P[294]{
   GP1:
	UF : 1, UT : 1,		CONFIG : 'N U T, 0, 0, 0',
	X =  2685.132  mm,	Y =   201.280  mm,	Z =   305.695  mm,
	W =    -3.830 deg,	P =   -10.878 deg,	R =   -17.892 deg
   GP2:
	UF : 1, UT : 1,
	J1=    90.000 deg,	J2=   135.000 deg
};
P[295]{
   GP1:
	UF : 1, UT : 1,		CONFIG : 'N U T, 0, 0, 0',
	X =  2753.412  mm,	Y =   160.459  mm,	Z =   180.671  mm,
	W =     2.791 deg,	P =    -7.674 deg,	R =   -18.462 deg
   GP2:
	UF : 1, UT : 1,
	J1=    90.000 deg,	J2=   135.000 deg
};
P[296]{
   GP1:
	UF : 1, UT : 1,		CONFIG : 'N U T, 0, 0, 0',
	X =  2867.805  mm,	Y =   160.634  mm,	Z =   182.471  mm,
	W =     9.502 deg,	P =   -26.582 deg,	R =   -20.495 deg
   GP2:
	UF : 1, UT : 1,
	J1=    89.999 deg,	J2=   135.000 deg
};
P[297]{
   GP1:
	UF : 1, UT : 1,		CONFIG : 'N U T, 0, 0, 0',
	X =  2663.741  mm,	Y =   157.782  mm,	Z =   292.643  mm,
	W =    13.374 deg,	P =   -35.036 deg,	R =   -22.495 deg
   GP2:
	UF : 1, UT : 1,
	J1=    90.000 deg,	J2=   135.000 deg
};
P[298]{
   GP1:
	UF : 1, UT : 1,		CONFIG : 'N U T, 0, 0, 0',
	X =  2363.741  mm,	Y =   272.782  mm,	Z =   292.643  mm,
	W =     -.090 deg,	P =    -5.498 deg,	R =      .950 deg
   GP2:
	UF : 1, UT : 1,
	J1=    90.000 deg,	J2=   135.000 deg
};
P[299]{
   GP1:
	UF : 1, UT : 1,		CONFIG : 'N U T, 0, 0, 0',
	X =  2378.956  mm,	Y =   265.120  mm,	Z =    86.366  mm,
	W =     1.850 deg,	P =     -.182 deg,	R =      .942 deg
   GP2:
	UF : 1, UT : 1,
	J1=    90.000 deg,	J2=   135.000 deg
};
P[300]{
   GP1:
	UF : 1, UT : 1,		CONFIG : 'N U T, 0, 0, 0',
	X =  2754.391  mm,	Y =   263.612  mm,	Z =    86.366  mm,
	W =     1.733 deg,	P =    -7.250 deg,	R =      .949 deg
   GP2:
	UF : 1, UT : 1,
	J1=    90.000 deg,	J2=   135.000 deg
};
P[301]{
   GP1:
	UF : 1, UT : 1,		CONFIG : 'N U T, 0, 0, 0',
	X =  2718.394  mm,	Y =   243.937  mm,	Z =   215.203  mm,
	W =     -.140 deg,	P =    -8.465 deg,	R =      .956 deg
   GP2:
	UF : 1, UT : 1,
	J1=    90.000 deg,	J2=   135.000 deg
};
P[302]{
   GP1:
	UF : 1, UT : 1,		CONFIG : 'N U T, 0, 0, 0',
	X =  2303.751  mm,	Y =   260.223  mm,	Z =   215.203  mm,
	W =     -.140 deg,	P =    -8.465 deg,	R =      .956 deg
   GP2:
	UF : 1, UT : 1,
	J1=    90.000 deg,	J2=   135.000 deg
};
P[303]{
   GP1:
	UF : 1, UT : 1,		CONFIG : 'N U T, 0, 0, 0',
	X =  1858.037  mm,	Y =   423.080  mm,	Z =   600.917  mm,
	W =     -.140 deg,	P =    -8.465 deg,	R =   -19.002 deg
   GP2:
	UF : 1, UT : 1,
	J1=    90.000 deg,	J2=   135.000 deg
};
P[304]{
   GP1:
	UF : 1, UT : 1,		CONFIG : 'N U T, 0, 0, 0',
	X =  1858.037  mm,	Y =   423.080  mm,	Z =   369.489  mm,
	W =    39.110 deg,	P =     2.688 deg,	R =   -82.797 deg
   GP2:
	UF : 1, UT : 1,
	J1=    90.000 deg,	J2=    90.000 deg
};
P[305]{
   GP1:
	UF : 1, UT : 1,		CONFIG : 'N U T, 0, 0, 0',
	X =  2035.037  mm,	Y =    99.189  mm,	Z =    92.489  mm,
	W =    39.110 deg,	P =     2.688 deg,	R =   -82.797 deg
   GP2:
	UF : 1, UT : 1,
	J1=    90.000 deg,	J2=    90.000 deg
};
P[306]{
   GP1:
	UF : 1, UT : 1,		CONFIG : 'N U T, 0, 0, 0',
	X =  2068.312  mm,	Y =   107.394  mm,	Z =   -18.582  mm,
	W =    37.933 deg,	P =    17.387 deg,	R =   -97.672 deg
   GP2:
	UF : 1, UT : 1,
	J1=    90.000 deg,	J2=    90.000 deg
};
P[307]{
   GP1:
	UF : 1, UT : 1,		CONFIG : 'N U T, 0, 0, 0',
	X =  2109.723  mm,	Y =    72.505  mm,	Z =   -21.222  mm,
	W =    37.933 deg,	P =    17.387 deg,	R =  -104.287 deg
   GP2:
	UF : 1, UT : 1,
	J1=    90.000 deg,	J2=    90.000 deg
};
P[308]{
   GP1:
	UF : 1, UT : 1,		CONFIG : 'N U T, 0, 0, -1',
	X =  2115.592  mm,	Y =    62.473  mm,	Z =   -16.026  mm,
	W =    44.181 deg,	P =    21.261 deg,	R =  -126.963 deg
   GP2:
	UF : 1, UT : 1,
	J1=    90.000 deg,	J2=    90.000 deg
};
P[309]{
   GP1:
	UF : 1, UT : 1,		CONFIG : 'N U T, 0, 0, -1',
	X =  2027.388  mm,	Y =   105.837  mm,	Z =    81.683  mm,
	W =    40.362 deg,	P =    21.867 deg,	R =  -139.995 deg
   GP2:
	UF : 1, UT : 1,
	J1=    90.000 deg,	J2=    90.000 deg
};
P[310]{
   GP1:
	UF : 1, UT : 1,		CONFIG : 'N U T, 0, 0, 0',
	X =  1658.817  mm,	Y =   448.694  mm,	Z =    81.684  mm,
	W =   -42.959 deg,	P =    14.926 deg,	R =    16.534 deg
   GP2:
	UF : 1, UT : 1,
	J1=    90.000 deg,	J2=    90.000 deg
};
P[311]{
   GP1:
	UF : 1, UT : 1,		CONFIG : 'N U T, 0, 0, 0',
	X =  1681.875  mm,	Y =   114.694  mm,	Z =    81.683  mm,
	W =   -42.959 deg,	P =    14.926 deg,	R =    16.534 deg
   GP2:
	UF : 1, UT : 1,
	J1=    90.000 deg,	J2=    90.000 deg
};
P[312]{
   GP1:
	UF : 1, UT : 1,		CONFIG : 'N U T, 0, 0, 0',
	X =  1685.743  mm,	Y =    59.810  mm,	Z =   -17.917  mm,
	W =   -42.807 deg,	P =    15.441 deg,	R =    16.037 deg
   GP2:
	UF : 1, UT : 1,
	J1=    90.000 deg,	J2=    90.000 deg
};
P[313]{
   GP1:
	UF : 1, UT : 1,		CONFIG : 'N U T, 0, 0, 0',
	X =  1652.429  mm,	Y =    58.946  mm,	Z =   -19.364  mm,
	W =   -42.810 deg,	P =    15.442 deg,	R =    16.034 deg
   GP2:
	UF : 1, UT : 1,
	J1=    90.000 deg,	J2=    90.000 deg
};
P[314]{
   GP1:
	UF : 1, UT : 1,		CONFIG : 'N U T, 0, 0, 0',
	X =  1640.987  mm,	Y =    56.683  mm,	Z =   -21.519  mm,
	W =   -42.181 deg,	P =    15.522 deg,	R =    -8.109 deg
   GP2:
	UF : 1, UT : 1,
	J1=    90.000 deg,	J2=    90.000 deg
};
P[315]{
   GP1:
	UF : 1, UT : 1,		CONFIG : 'N U T, 0, 0, 0',
	X =  1637.701  mm,	Y =    59.485  mm,	Z =   -19.665  mm,
	W =   -38.593 deg,	P =    25.218 deg,	R =   -16.905 deg
   GP2:
	UF : 1, UT : 1,
	J1=    90.000 deg,	J2=    90.000 deg
};
P[316]{
   GP1:
	UF : 1, UT : 1,		CONFIG : 'N U T, 0, 0, 0',
	X =  1608.736  mm,	Y =    83.348  mm,	Z =   -24.399  mm,
	W =   -38.593 deg,	P =    25.219 deg,	R =   -16.905 deg
   GP2:
	UF : 1, UT : 1,
	J1=    90.000 deg,	J2=    90.000 deg
};
P[317]{
   GP1:
	UF : 1, UT : 1,		CONFIG : 'N U T, 0, 0, 0',
	X =  1585.662  mm,	Y =   101.135  mm,	Z =   -21.859  mm,
	W =   -45.000 deg,	P =    -3.170 deg,	R =      .426 deg
   GP2:
	UF : 1, UT : 1,
	J1=    90.000 deg,	J2=    90.000 deg
};
P[318]{
   GP1:
	UF : 1, UT : 1,		CONFIG : 'N U T, 0, 0, 0',
	X =  1556.810  mm,	Y =    69.060  mm,	Z =   -21.622  mm,
	W =   -45.449 deg,	P =    19.944 deg,	R =    98.982 deg
   GP2:
	UF : 1, UT : 1,
	J1=    90.000 deg,	J2=    90.000 deg
};
P[319]{
   GP1:
	UF : 1, UT : 1,		CONFIG : 'N U T, 0, 0, 0',
	X =  1551.240  mm,	Y =    28.811  mm,	Z =   -19.922  mm,
	W =   -45.337 deg,	P =    20.062 deg,	R =    97.887 deg
   GP2:
	UF : 1, UT : 1,
	J1=    90.000 deg,	J2=    90.000 deg
};
P[320]{
   GP1:
	UF : 1, UT : 1,		CONFIG : 'N U T, 0, 0, 0',
	X =  1551.443  mm,	Y =    22.198  mm,	Z =   -20.367  mm,
	W =   -45.343 deg,	P =    20.068 deg,	R =    97.646 deg
   GP2:
	UF : 1, UT : 1,
	J1=    90.000 deg,	J2=    90.000 deg
};
P[321]{
   GP1:
	UF : 1, UT : 1,		CONFIG : 'N U T, 0, 0, 0',
	X =  1549.407  mm,	Y =    21.768  mm,	Z =   -17.950  mm,
	W =   -41.210 deg,	P =    19.947 deg,	R =    34.862 deg
   GP2:
	UF : 1, UT : 1,
	J1=    90.000 deg,	J2=    90.000 deg
};
P[322]{
   GP1:
	UF : 1, UT : 1,		CONFIG : 'N U T, 0, 0, 0',
	X =  1540.684  mm,	Y =    20.490  mm,	Z =   -17.846  mm,
	W =   -41.215 deg,	P =    19.945 deg,	R =    34.866 deg
   GP2:
	UF : 1, UT : 1,
	J1=    90.000 deg,	J2=    90.000 deg
};
P[323]{
   GP1:
	UF : 1, UT : 1,		CONFIG : 'N U T, 0, 0, 0',
	X =  1231.677  mm,	Y =   199.953  mm,	Z =   178.712  mm,
	W =   -41.215 deg,	P =    19.944 deg,	R =    40.052 deg
   GP2:
	UF : 1, UT : 1,
	J1=    90.000 deg,	J2=    90.000 deg
};
P[324]{
   GP1:
	UF : 1, UT : 1,		CONFIG : 'N U T, 0, 0, 0',
	X =   877.425  mm,	Y =  1334.354  mm,	Z =    94.527  mm,
	W =     -.178 deg,	P =    -1.186 deg,	R =    26.509 deg
   GP2:
	UF : 1, UT : 1,
	J1=    90.000 deg,	J2=    90.000 deg
};
P[325]{
   GP1:
	UF : 1, UT : 1,		CONFIG : 'N U T, 0, 0, 0',
	X =  2712.426  mm,	Y =  1334.354  mm,	Z =    94.527  mm,
	W =     -.178 deg,	P =    -1.186 deg,	R =    26.509 deg
   GP2:
	UF : 1, UT : 1,
	J1=    90.000 deg,	J2=    90.000 deg
};
P[326]{
   GP1:
	UF : 1, UT : 1,		CONFIG : 'N U T, 0, 0, 0',
	X =  2866.453  mm,	Y =  1420.346  mm,	Z =   -11.619  mm,
	W =     -.178 deg,	P =    -1.186 deg,	R =    26.508 deg
   GP2:
	UF : 1, UT : 1,
	J1=    90.000 deg,	J2=    90.000 deg
};
P[327]{
   GP1:
	UF : 1, UT : 1,		CONFIG : 'N U T, 0, 0, 0',
	X =  2866.454  mm,	Y =  1403.775  mm,	Z =   -11.619  mm,
	W =     -.178 deg,	P =    -1.186 deg,	R =    26.508 deg
   GP2:
	UF : 1, UT : 1,
	J1=    90.000 deg,	J2=    90.000 deg
};
P[328]{
   GP1:
	UF : 1, UT : 1,		CONFIG : 'N U T, 0, 0, 0',
	X =  2851.597  mm,	Y =  1403.775  mm,	Z =   -11.619  mm,
	W =     -.178 deg,	P =    -1.186 deg,	R =    26.508 deg
   GP2:
	UF : 1, UT : 1,
	J1=    90.000 deg,	J2=    90.000 deg
};
P[329]{
   GP1:
	UF : 1, UT : 1,		CONFIG : 'N U T, 0, 0, 0',
	X =  2851.596  mm,	Y =  1403.775  mm,	Z =    -7.333  mm,
	W =     -.178 deg,	P =    -1.186 deg,	R =    26.508 deg
   GP2:
	UF : 1, UT : 1,
	J1=    90.000 deg,	J2=    90.000 deg
};
P[330]{
   GP1:
	UF : 1, UT : 1,		CONFIG : 'N U T, 0, 0, 0',
	X =  2851.355  mm,	Y =  1420.068  mm,	Z =   -11.543  mm,
	W =     -.178 deg,	P =    -1.186 deg,	R =    26.509 deg
   GP2:
	UF : 1, UT : 1,
	J1=    90.000 deg,	J2=    90.000 deg
};
P[331]{
   GP1:
	UF : 1, UT : 1,		CONFIG : 'N U T, 0, 0, 0',
	X =  2851.355  mm,	Y =  1420.068  mm,	Z =    -7.258  mm,
	W =     -.178 deg,	P =    -1.186 deg,	R =    26.509 deg
   GP2:
	UF : 1, UT : 1,
	J1=    90.000 deg,	J2=    90.000 deg
};
P[332]{
   GP1:
	UF : 1, UT : 1,		CONFIG : 'N U T, 0, 0, 0',
	X =  2712.426  mm,	Y =  1334.354  mm,	Z =    94.527  mm,
	W =     -.178 deg,	P =    -1.186 deg,	R =    26.509 deg
   GP2:
	UF : 1, UT : 1,
	J1=    90.000 deg,	J2=    90.000 deg
};
P[333]{
   GP1:
	UF : 1, UT : 1,		CONFIG : 'N U T, 0, 0, 0',
	X =   877.425  mm,	Y =  1334.354  mm,	Z =    94.527  mm,
	W =     -.178 deg,	P =    -1.186 deg,	R =    26.509 deg
   GP2:
	UF : 1, UT : 1,
	J1=    90.000 deg,	J2=    90.000 deg
};
P[334]{
   GP1:
	UF : 1, UT : 1,		CONFIG : 'N U T, 0, 0, 0',
	X =  1097.392  mm,	Y =  -178.047  mm,	Z =   178.712  mm,
	W =   -34.745 deg,	P =    30.619 deg,	R =   119.475 deg
   GP2:
	UF : 1, UT : 1,
	J1=    90.000 deg,	J2=    90.000 deg
};
P[335]{
   GP1:
	UF : 1, UT : 1,		CONFIG : 'N U T, 0, 0, 0',
	X =  1587.677  mm,	Y =  -226.342  mm,	Z =    50.712  mm,
	W =   -34.744 deg,	P =    30.618 deg,	R =   128.397 deg
   GP2:
	UF : 1, UT : 1,
	J1=    90.000 deg,	J2=    90.000 deg
};
P[336]{
   GP1:
	UF : 1, UT : 1,		CONFIG : 'N U T, 0, 0, 1',
	X =  1651.536  mm,	Y =  -219.100  mm,	Z =   -19.888  mm,
	W =   -32.939 deg,	P =    29.350 deg,	R =   129.300 deg
   GP2:
	UF : 1, UT : 1,
	J1=    90.000 deg,	J2=    90.000 deg
};
P[337]{
   GP1:
	UF : 1, UT : 1,		CONFIG : 'N U T, 0, 0, 1',
	X =  1652.465  mm,	Y =    20.682  mm,	Z =   -20.854  mm,
	W =   -34.233 deg,	P =    30.069 deg,	R =   141.356 deg
   GP2:
	UF : 1, UT : 1,
	J1=    90.000 deg,	J2=    90.000 deg
};
P[338]{
   GP1:
	UF : 1, UT : 1,		CONFIG : 'N U T, 0, 0, 1',
	X =  1473.582  mm,	Y =   -83.067  mm,	Z =   190.803  mm,
	W =   -34.742 deg,	P =    30.617 deg,	R =   153.799 deg
   GP2:
	UF : 1, UT : 1,
	J1=    90.000 deg,	J2=    90.000 deg
};
P[339]{
   GP1:
	UF : 1, UT : 1,		CONFIG : 'N U T, 0, 0, 0',
	X =  1333.582  mm,	Y =  -300.066  mm,	Z =   190.803  mm,
	W =    44.863 deg,	P =    -3.871 deg,	R =     -.364 deg
   GP2:
	UF : 1, UT : 1,
	J1=    90.000 deg,	J2=    90.000 deg
};
P[340]{
   GP1:
	UF : 1, UT : 1,		CONFIG : 'N U T, 0, 0, 0',
	X =  2404.583  mm,	Y =  -249.066  mm,	Z =    43.803  mm,
	W =    42.099 deg,	P =    -2.376 deg,	R =   -15.667 deg
   GP2:
	UF : 1, UT : 1,
	J1=    90.000 deg,	J2=    90.000 deg
};
P[341]{
   GP1:
	UF : 1, UT : 1,		CONFIG : 'N U T, 0, 0, 0',
	X =  2351.061  mm,	Y =  -179.371  mm,	Z =   -13.077  mm,
	W =    44.587 deg,	P =     6.899 deg,	R =    -6.951 deg
   GP2:
	UF : 1, UT : 1,
	J1=    90.000 deg,	J2=    90.000 deg
};
P[342]{
   GP1:
	UF : 1, UT : 1,		CONFIG : 'N U T, 0, 0, 0',
	X =  2518.615  mm,	Y =  -178.195  mm,	Z =   -13.758  mm,
	W =    44.582 deg,	P =     6.892 deg,	R =    -6.941 deg
   GP2:
	UF : 1, UT : 1,
	J1=    90.000 deg,	J2=    90.000 deg
};
P[343]{
   GP1:
	UF : 1, UT : 1,		CONFIG : 'N U T, 0, 0, 0',
	X =  2517.065  mm,	Y =  -219.497  mm,	Z =    58.957  mm,
	W =    44.580 deg,	P =     6.891 deg,	R =   -21.154 deg
   GP2:
	UF : 1, UT : 1,
	J1=    90.000 deg,	J2=    90.000 deg
};
P[344]{
   GP1:
	UF : 1, UT : 1,		CONFIG : 'N U T, 0, 0, 0',
	X =  2344.098  mm,	Y =  -219.497  mm,	Z =    58.957  mm,
	W =    44.580 deg,	P =     6.891 deg,	R =   -21.154 deg
   GP2:
	UF : 1, UT : 1,
	J1=    90.000 deg,	J2=    90.000 deg
};
P[345]{
   GP1:
	UF : 1, UT : 1,		CONFIG : 'N U T, 0, 0, 0',
	X =  2344.098  mm,	Y =  -132.497  mm,	Z =    58.956  mm,
	W =    44.580 deg,	P =     6.891 deg,	R =   -21.154 deg
   GP2:
	UF : 1, UT : 1,
	J1=    90.000 deg,	J2=    90.000 deg
};
P[346]{
   GP1:
	UF : 1, UT : 1,		CONFIG : 'N U T, 0, 0, 0',
	X =  2352.052  mm,	Y =   -90.042  mm,	Z =   -15.707  mm,
	W =    43.242 deg,	P =    13.891 deg,	R =   -18.605 deg
   GP2:
	UF : 1, UT : 1,
	J1=    90.000 deg,	J2=    90.000 deg
};
P[347]{
   GP1:
	UF : 1, UT : 1,		CONFIG : 'N U T, 0, 0, 0',
	X =  2404.409  mm,	Y =   -89.953  mm,	Z =   -14.975  mm,
	W =    43.244 deg,	P =    13.890 deg,	R =   -18.607 deg
   GP2:
	UF : 1, UT : 1,
	J1=    90.000 deg,	J2=    90.000 deg
};
P[348]{
   GP1:
	UF : 1, UT : 1,		CONFIG : 'N U T, 0, 0, 0',
	X =  2423.248  mm,	Y =   -92.540  mm,	Z =    -8.646  mm,
	W =    42.728 deg,	P =    13.810 deg,	R =   -51.889 deg
   GP2:
	UF : 1, UT : 1,
	J1=    89.998 deg,	J2=    90.000 deg
};
P[349]{
   GP1:
	UF : 1, UT : 1,		CONFIG : 'N U T, 0, 0, 0',
	X =  2344.098  mm,	Y =  -132.497  mm,	Z =    58.956  mm,
	W =    44.580 deg,	P =     6.891 deg,	R =   -21.154 deg
   GP2:
	UF : 1, UT : 1,
	J1=    90.000 deg,	J2=    90.000 deg
};
P[350]{
   GP1:
	UF : 1, UT : 1,		CONFIG : 'N U T, 0, 0, 0',
	X =  1084.097  mm,	Y =  -132.497  mm,	Z =   115.956  mm,
	W =    46.380 deg,	P =     2.235 deg,	R =    13.463 deg
   GP2:
	UF : 1, UT : 1,
	J1=    90.000 deg,	J2=    90.000 deg
};
P[351]{
   GP1:
	UF : 1, UT : 1,		CONFIG : 'N U T, 0, 0, 0',
	X =  1084.097  mm,	Y =  -132.497  mm,	Z =  1093.099  mm,
	W =    23.155 deg,	P =    41.431 deg,	R =   -41.534 deg
   GP2:
	UF : 1, UT : 1,
	J1=    90.000 deg,	J2=    90.000 deg
};
P[352]{
   GP1:
	UF : 1, UT : 1,		CONFIG : 'N U T, 0, 0, 0',
	X =   922.816  mm,	Y =    -9.239  mm,	Z =  2168.306  mm,
	W =     -.010 deg,	P =   -45.000 deg,	R =     0.000 deg
   GP2:
	UF : 1, UT : 1,
	J1=   -90.000 deg,	J2=   -90.000 deg
};
P[353]{
   GP1:
	UF : 1, UT : 1,		CONFIG : 'N U T, 0, 0, 0',
	X =   922.816  mm,	Y =    -9.239  mm,	Z =  1240.448  mm,
	W =    39.867 deg,	P =   -22.888 deg,	R =   -65.014 deg
   GP2:
	UF : 1, UT : 1,
	J1=   -90.000 deg,	J2=   -90.000 deg
};
P[354]{
   GP1:
	UF : 1, UT : 1,		CONFIG : 'N U T, 0, 0, 0',
	X =  1630.173  mm,	Y =   470.761  mm,	Z =   907.448  mm,
	W =    39.867 deg,	P =   -22.888 deg,	R =   -65.014 deg
   GP2:
	UF : 1, UT : 1,
	J1=   -90.000 deg,	J2=   -90.000 deg
};
P[355]{
   GP1:
	UF : 1, UT : 1,		CONFIG : 'N U T, 0, 0, 0',
	X =  1684.563  mm,	Y =   458.656  mm,	Z =   830.406  mm,
	W =    39.866 deg,	P =   -22.888 deg,	R =   -65.013 deg
   GP2:
	UF : 1, UT : 1,
	J1=   -90.000 deg,	J2=   -90.000 deg
};
P[356]{
   GP1:
	UF : 1, UT : 1,		CONFIG : 'N U T, 0, 0, 0',
	X =  1685.493  mm,	Y =   473.679  mm,	Z =   828.230  mm,
	W =    39.866 deg,	P =   -22.887 deg,	R =   -65.013 deg
   GP2:
	UF : 1, UT : 1,
	J1=   -90.000 deg,	J2=   -90.000 deg
};
P[357]{
   GP1:
	UF : 1, UT : 1,		CONFIG : 'N U T, 0, 0, 0',
	X =  1685.563  mm,	Y =   480.822  mm,	Z =   829.093  mm,
	W =    39.867 deg,	P =   -22.888 deg,	R =   -69.837 deg
   GP2:
	UF : 1, UT : 1,
	J1=   -90.000 deg,	J2=   -90.000 deg
};
P[358]{
   GP1:
	UF : 1, UT : 1,		CONFIG : 'N U T, 0, 0, 0',
	X =  1687.491  mm,	Y =   484.680  mm,	Z =   827.711  mm,
	W =    39.867 deg,	P =   -22.888 deg,	R =   -70.971 deg
   GP2:
	UF : 1, UT : 1,
	J1=   -90.000 deg,	J2=   -90.000 deg
};
P[359]{
   GP1:
	UF : 1, UT : 1,		CONFIG : 'N U T, 0, 0, 0',
	X =  1708.839  mm,	Y =   554.633  mm,	Z =   827.423  mm,
	W =    39.871 deg,	P =   -22.884 deg,	R =   -70.976 deg
   GP2:
	UF : 1, UT : 1,
	J1=   -90.000 deg,	J2=   -90.000 deg
};
P[360]{
   GP1:
	UF : 1, UT : 1,		CONFIG : 'N U T, 0, 0, 0',
	X =  1711.676  mm,	Y =   557.080  mm,	Z =   826.531  mm,
	W =    39.870 deg,	P =   -22.884 deg,	R =   -74.846 deg
   GP2:
	UF : 1, UT : 1,
	J1=   -90.000 deg,	J2=   -90.000 deg
};
P[361]{
   GP1:
	UF : 1, UT : 1,		CONFIG : 'N U T, 0, 0, 0',
	X =  1712.809  mm,	Y =   560.962  mm,	Z =   826.801  mm,
	W =    39.866 deg,	P =   -22.883 deg,	R =   -82.536 deg
   GP2:
	UF : 1, UT : 1,
	J1=   -90.000 deg,	J2=   -90.000 deg
};
P[362]{
   GP1:
	UF : 1, UT : 1,		CONFIG : 'N U T, 0, 0, 0',
	X =  1845.680  mm,	Y =   825.086  mm,	Z =   832.601  mm,
	W =    14.309 deg,	P =   -43.038 deg,	R =   -40.623 deg
   GP2:
	UF : 1, UT : 1,
	J1=   -89.991 deg,	J2=   -89.999 deg
};
P[363]{
   GP1:
	UF : 1, UT : 1,		CONFIG : 'N U T, 0, 0, 0',
	X =  1719.210  mm,	Y =   890.070  mm,	Z =   992.766  mm,
	W =   -20.210 deg,	P =   -41.106 deg,	R =     1.246 deg
   GP2:
	UF : 1, UT : 1,
	J1=   -90.000 deg,	J2=   -90.000 deg
};
P[364]{
   GP1:
	UF : 1, UT : 1,		CONFIG : 'N U T, 0, 0, 0',
	X =  1696.710  mm,	Y =   336.928  mm,	Z =   932.155  mm,
	W =    42.022 deg,	P =   -15.891 deg,	R =   -33.571 deg
   GP2:
	UF : 1, UT : 1,
	J1=   -90.000 deg,	J2=   -90.000 deg
};
P[365]{
   GP1:
	UF : 1, UT : 1,		CONFIG : 'N U T, 0, 0, 0',
	X =  1698.333  mm,	Y =   426.907  mm,	Z =   830.357  mm,
	W =    43.050 deg,	P =   -14.373 deg,	R =   -45.079 deg
   GP2:
	UF : 1, UT : 1,
	J1=   -90.000 deg,	J2=   -90.000 deg
};
P[366]{
   GP1:
	UF : 1, UT : 1,		CONFIG : 'N U T, 0, 0, 0',
	X =  1839.303  mm,	Y =   266.347  mm,	Z =   829.243  mm,
	W =    43.053 deg,	P =   -14.369 deg,	R =   -45.082 deg
   GP2:
	UF : 1, UT : 1,
	J1=   -90.000 deg,	J2=   -90.000 deg
};
P[367]{
   GP1:
	UF : 1, UT : 1,		CONFIG : 'N U T, 0, 0, 0',
	X =  1847.539  mm,	Y =   258.366  mm,	Z =   830.212  mm,
	W =    43.049 deg,	P =   -14.375 deg,	R =   -42.871 deg
   GP2:
	UF : 1, UT : 1,
	J1=   -90.000 deg,	J2=   -90.000 deg
};
P[368]{
   GP1:
	UF : 1, UT : 1,		CONFIG : 'N U T, 0, 0, 0',
	X =  1859.538  mm,	Y =   247.937  mm,	Z =   830.256  mm,
	W =    43.049 deg,	P =   -14.375 deg,	R =   -40.829 deg
   GP2:
	UF : 1, UT : 1,
	J1=   -90.000 deg,	J2=   -90.000 deg
};
P[369]{
   GP1:
	UF : 1, UT : 1,		CONFIG : 'N U T, 0, 0, 0',
	X =  1923.179  mm,	Y =   200.865  mm,	Z =   829.012  mm,
	W =    43.049 deg,	P =   -14.374 deg,	R =   -40.829 deg
   GP2:
	UF : 1, UT : 1,
	J1=   -90.000 deg,	J2=   -90.000 deg
};
P[370]{
   GP1:
	UF : 1, UT : 1,		CONFIG : 'N U T, 0, 0, 0',
	X =  1870.572  mm,	Y =   165.642  mm,	Z =   951.351  mm,
	W =    58.350 deg,	P =   -26.173 deg,	R =   -73.280 deg
   GP2:
	UF : 1, UT : 1,
	J1=   -90.000 deg,	J2=   -90.000 deg
};
P[371]{
   GP1:
	UF : 1, UT : 1,		CONFIG : 'N U T, 0, 0, 0',
	X =   849.429  mm,	Y =   203.927  mm,	Z =   951.351  mm,
	W =    58.350 deg,	P =   -26.173 deg,	R =   -73.280 deg
   GP2:
	UF : 1, UT : 1,
	J1=   -90.000 deg,	J2=   -90.000 deg
};
P[372]{
   GP1:
	UF : 1, UT : 1,		CONFIG : 'N U T, 0, 0, 0',
	X =   556.988  mm,	Y =    -6.143  mm,	Z =  1500.654  mm,
	W =     -.033 deg,	P =    22.090 deg,	R =      .044 deg
   GP2:
	UF : 1, UT : 1,
	J1=   -70.000 deg,	J2=    45.000 deg
};
P[373]{
   GP1:
	UF : 1, UT : 1,		CONFIG : 'N U T, 0, 0, 0',
	X =   556.950  mm,	Y =    -6.098  mm,	Z =  1500.653  mm,
	W =     -.030 deg,	P =    22.091 deg,	R =      .051 deg
   GP2:
	UF : 1, UT : 1,
	J1=   -90.000 deg,	J2=    90.000 deg
};
P[374]{
   GP1:
	UF : 1, UT : 1,		CONFIG : 'N U T, 0, 0, 0',
	X =  1449.587  mm,	Y =  -481.240  mm,	Z =   957.304  mm,
	W =     -.010 deg,	P =   -46.549 deg,	R =     0.000 deg
   GP2:
	UF : 1, UT : 1,
	J1=   -90.000 deg,	J2=    90.000 deg
};
P[375]{
   GP1:
	UF : 1, UT : 1,		CONFIG : 'N U T, 0, 0, 0',
	X =  1660.516  mm,	Y =  -481.240  mm,	Z =   876.304  mm,
	W =   -29.059 deg,	P =   -38.116 deg,	R =    41.980 deg
   GP2:
	UF : 1, UT : 1,
	J1=   -90.000 deg,	J2=    90.000 deg
};
P[376]{
   GP1:
	UF : 1, UT : 1,		CONFIG : 'N U T, 0, 0, 0',
	X =  1678.881  mm,	Y =  -469.975  mm,	Z =   829.150  mm,
	W =   -28.314 deg,	P =   -37.469 deg,	R =    36.647 deg
   GP2:
	UF : 1, UT : 1,
	J1=   -90.000 deg,	J2=    90.000 deg
};
P[377]{
   GP1:
	UF : 1, UT : 1,		CONFIG : 'N U T, 0, 0, 0',
	X =  1682.926  mm,	Y =  -487.189  mm,	Z =   826.659  mm,
	W =   -28.322 deg,	P =   -37.469 deg,	R =    36.650 deg
   GP2:
	UF : 1, UT : 1,
	J1=   -90.000 deg,	J2=    90.000 deg
};
P[378]{
   GP1:
	UF : 1, UT : 1,		CONFIG : 'N U T, 0, 0, 0',
	X =  1682.542  mm,	Y =  -491.734  mm,	Z =   828.424  mm,
	W =   -28.334 deg,	P =   -37.464 deg,	R =    39.731 deg
   GP2:
	UF : 1, UT : 1,
	J1=   -90.000 deg,	J2=    90.000 deg
};
P[379]{
   GP1:
	UF : 1, UT : 1,		CONFIG : 'N U T, 0, 0, 0',
	X =  1683.217  mm,	Y =  -494.546  mm,	Z =   827.297  mm,
	W =   -28.322 deg,	P =   -37.469 deg,	R =    41.171 deg
   GP2:
	UF : 1, UT : 1,
	J1=   -90.000 deg,	J2=    90.000 deg
};
P[380]{
   GP1:
	UF : 1, UT : 1,		CONFIG : 'N U T, 0, 0, 0',
	X =  1707.638  mm,	Y =  -565.332  mm,	Z =   825.835  mm,
	W =   -28.322 deg,	P =   -37.469 deg,	R =    41.171 deg
   GP2:
	UF : 1, UT : 1,
	J1=   -90.000 deg,	J2=    90.000 deg
};
P[381]{
   GP1:
	UF : 1, UT : 1,		CONFIG : 'N U T, 0, 0, 0',
	X =  1709.098  mm,	Y =  -569.548  mm,	Z =   825.685  mm,
	W =   -28.322 deg,	P =   -37.469 deg,	R =    48.505 deg
   GP2:
	UF : 1, UT : 1,
	J1=   -90.000 deg,	J2=    90.000 deg
};
P[382]{
   GP1:
	UF : 1, UT : 1,		CONFIG : 'N U T, 0, 0, 0',
	X =  1713.633  mm,	Y =  -574.840  mm,	Z =   824.222  mm,
	W =   -28.328 deg,	P =   -37.465 deg,	R =    55.403 deg
   GP2:
	UF : 1, UT : 1,
	J1=   -90.000 deg,	J2=    90.000 deg
};
P[383]{
   GP1:
	UF : 1, UT : 1,		CONFIG : 'N U T, 0, 0, 0',
	X =  1842.146  mm,	Y =  -829.157  mm,	Z =   829.639  mm,
	W =   -28.322 deg,	P =   -37.469 deg,	R =    50.636 deg
   GP2:
	UF : 1, UT : 1,
	J1=   -90.000 deg,	J2=    90.000 deg
};
P[384]{
   GP1:
	UF : 1, UT : 1,		CONFIG : 'N U T, 0, 0, 0',
	X =  1612.442  mm,	Y =  -863.138  mm,	Z =   905.385  mm,
	W =   -20.245 deg,	P =   -41.090 deg,	R =    57.299 deg
   GP2:
	UF : 1, UT : 1,
	J1=   -90.000 deg,	J2=    90.000 deg
};
P[385]{
   GP1:
	UF : 1, UT : 1,		CONFIG : 'N U T, 0, 0, 0',
	X =  1612.442  mm,	Y =  -365.996  mm,	Z =   905.386  mm,
	W =   -53.336 deg,	P =     2.108 deg,	R =    49.603 deg
   GP2:
	UF : 1, UT : 1,
	J1=   -90.000 deg,	J2=    90.000 deg
};
P[386]{
   GP1:
	UF : 1, UT : 1,		CONFIG : 'N U T, 0, 0, 0',
	X =  1690.304  mm,	Y =  -437.670  mm,	Z =   830.884  mm,
	W =   -39.460 deg,	P =    -8.334 deg,	R =    42.657 deg
   GP2:
	UF : 1, UT : 1,
	J1=   -90.000 deg,	J2=    90.000 deg
};
P[387]{
   GP1:
	UF : 1, UT : 1,		CONFIG : 'N U T, 0, 0, 0',
	X =  1836.271  mm,	Y =  -275.564  mm,	Z =   827.815  mm,
	W =   -39.460 deg,	P =    -8.334 deg,	R =    42.657 deg
   GP2:
	UF : 1, UT : 1,
	J1=   -90.000 deg,	J2=    90.000 deg
};
P[388]{
   GP1:
	UF : 1, UT : 1,		CONFIG : 'N U T, 0, 0, 0',
	X =  1848.380  mm,	Y =  -264.272  mm,	Z =   828.029  mm,
	W =   -39.460 deg,	P =    -8.334 deg,	R =    38.620 deg
   GP2:
	UF : 1, UT : 1,
	J1=   -90.000 deg,	J2=    90.000 deg
};
P[389]{
   GP1:
	UF : 1, UT : 1,		CONFIG : 'N U T, 0, 0, 0',
	X =  1862.737  mm,	Y =  -253.785  mm,	Z =   829.403  mm,
	W =   -39.460 deg,	P =    -8.334 deg,	R =    41.372 deg
   GP2:
	UF : 1, UT : 1,
	J1=   -90.000 deg,	J2=    90.000 deg
};
P[390]{
   GP1:
	UF : 1, UT : 1,		CONFIG : 'N U T, 0, 0, 0',
	X =  1935.611  mm,	Y =  -199.637  mm,	Z =   827.419  mm,
	W =   -39.460 deg,	P =    -8.334 deg,	R =    45.243 deg
   GP2:
	UF : 1, UT : 1,
	J1=   -90.000 deg,	J2=    90.000 deg
};
P[391]{
   GP1:
	UF : 1, UT : 1,		CONFIG : 'N U T, 0, 0, 0',
	X =  1827.763  mm,	Y =  -230.895  mm,	Z =   883.594  mm,
	W =   -54.261 deg,	P =    -6.374 deg,	R =    77.692 deg
   GP2:
	UF : 1, UT : 1,
	J1=   -90.000 deg,	J2=    90.000 deg
};
P[392]{
   GP1:
	UF : 1, UT : 1,		CONFIG : 'N U T, 0, 0, 0',
	X =   815.336  mm,	Y =  -406.109  mm,	Z =   870.736  mm,
	W =   -48.700 deg,	P =    -5.138 deg,	R =    77.361 deg
   GP2:
	UF : 1, UT : 1,
	J1=   -90.000 deg,	J2=    90.000 deg
};
P[393]{
   GP1:
	UF : 1, UT : 1,		CONFIG : 'N U T, 0, 0, 0',
	X =   922.816  mm,	Y =    -9.239  mm,	Z =  2168.306  mm,
	W =     -.010 deg,	P =   -45.000 deg,	R =     0.000 deg
   GP2:
	UF : 1, UT : 1,
	J1=    90.000 deg,	J2=    90.000 deg
};
P[394]{
   GP1:
	UF : 1, UT : 1,		CONFIG : 'N U T, 0, 0, 0',
	X =  2001.817  mm,	Y =    -9.239  mm,	Z =  1516.306  mm,
	W =     -.010 deg,	P =    45.000 deg,	R =    90.000 deg
   GP2:
	UF : 1, UT : 1,
	J1=    90.000 deg,	J2=    90.000 deg
};
P[395]{
   GP1:
	UF : 1, UT : 1,		CONFIG : 'N U T, 0, 0, 0',
	X =  2240.817  mm,	Y =   100.761  mm,	Z =   993.305  mm,
	W =     -.010 deg,	P =    44.999 deg,	R =    66.715 deg
   GP2:
	UF : 1, UT : 1,
	J1=    90.000 deg,	J2=    90.000 deg
};
P[396]{
   GP1:
	UF : 1, UT : 1,		CONFIG : 'N U T, 0, 0, 0',
	X =  2344.158  mm,	Y =   -61.498  mm,	Z =   837.144  mm,
	W =     4.733 deg,	P =    44.799 deg,	R =    66.706 deg
   GP2:
	UF : 1, UT : 1,
	J1=    90.000 deg,	J2=    90.000 deg
};
P[397]{
   GP1:
	UF : 1, UT : 1,		CONFIG : 'N U T, 0, 0, 0',
	X =  2404.770  mm,	Y =   -93.993  mm,	Z =   837.387  mm,
	W =     4.736 deg,	P =    44.803 deg,	R =    66.702 deg
   GP2:
	UF : 1, UT : 1,
	J1=    90.000 deg,	J2=    90.000 deg
};
P[398]{
   GP1:
	UF : 1, UT : 1,		CONFIG : 'N U T, 0, 0, 0',
	X =  2444.940  mm,	Y =   -30.095  mm,	Z =   912.480  mm,
	W =     4.736 deg,	P =    44.803 deg,	R =    66.702 deg
   GP2:
	UF : 1, UT : 1,
	J1=    90.000 deg,	J2=    90.000 deg
};
P[399]{
   GP1:
	UF : 1, UT : 1,		CONFIG : 'N U T, 0, 0, 0',
	X =  2429.507  mm,	Y =  -139.995  mm,	Z =   915.768  mm,
	W =   -19.426 deg,	P =    41.428 deg,	R =   -56.049 deg
   GP2:
	UF : 1, UT : 1,
	J1=    90.000 deg,	J2=    90.000 deg
};
P[400]{
   GP1:
	UF : 1, UT : 1,		CONFIG : 'N U T, 0, 0, 0',
	X =  2400.549  mm,	Y =  -120.824  mm,	Z =   838.185  mm,
	W =   -19.419 deg,	P =    41.428 deg,	R =   -56.052 deg
   GP2:
	UF : 1, UT : 1,
	J1=    90.000 deg,	J2=    90.000 deg
};
P[401]{
   GP1:
	UF : 1, UT : 1,		CONFIG : 'N U T, 0, 0, 0',
	X =  2411.665  mm,	Y =  -100.428  mm,	Z =   838.269  mm,
	W =   -19.426 deg,	P =    41.428 deg,	R =   -56.049 deg
   GP2:
	UF : 1, UT : 1,
	J1=    90.000 deg,	J2=    90.000 deg
};
P[402]{
   GP1:
	UF : 1, UT : 1,		CONFIG : 'N U T, 0, 0, 0',
	X =  2471.948  mm,	Y =  -129.877  mm,	Z =   908.172  mm,
	W =   -19.426 deg,	P =    41.428 deg,	R =   -56.049 deg
   GP2:
	UF : 1, UT : 1,
	J1=    90.000 deg,	J2=    90.000 deg
};
P[403]{
   GP1:
	UF : 1, UT : 1,		CONFIG : 'N U T, 0, 0, 0',
	X =  2171.268  mm,	Y =   -40.755  mm,	Z =   918.909  mm,
	W =    34.022 deg,	P =    31.444 deg,	R =   -66.610 deg
   GP2:
	UF : 1, UT : 1,
	J1=    90.000 deg,	J2=    90.000 deg
};
P[404]{
   GP1:
	UF : 1, UT : 1,		CONFIG : 'N U T, 0, 0, 0',
	X =  2329.816  mm,	Y =   -87.227  mm,	Z =   839.756  mm,
	W =    34.022 deg,	P =    31.444 deg,	R =   -66.610 deg
   GP2:
	UF : 1, UT : 1,
	J1=    90.000 deg,	J2=    90.000 deg
};
P[405]{
   GP1:
	UF : 1, UT : 1,		CONFIG : 'N U T, 0, 0, 0',
	X =  2393.327  mm,	Y =  -122.227  mm,	Z =   840.237  mm,
	W =    34.022 deg,	P =    31.444 deg,	R =   -66.610 deg
   GP2:
	UF : 1, UT : 1,
	J1=    90.000 deg,	J2=    90.000 deg
};
P[406]{
   GP1:
	UF : 1, UT : 1,		CONFIG : 'N U T, 0, 0, 0',
	X =  2236.242  mm,	Y =  -121.027  mm,	Z =   923.380  mm,
	W =    34.022 deg,	P =    31.444 deg,	R =   -66.610 deg
   GP2:
	UF : 1, UT : 1,
	J1=    90.000 deg,	J2=    90.000 deg
};
P[407]{
   GP1:
	UF : 1, UT : 1,		CONFIG : 'N U T, 0, 0, 0',
	X =  1125.569  mm,	Y =   539.568  mm,	Z =  1195.939  mm,
	W =    30.412 deg,	P =    23.153 deg,	R =   -68.803 deg
   GP2:
	UF : 1, UT : 1,
	J1=    90.000 deg,	J2=    90.000 deg
};
P[408]{
   GP1:
	UF : 1, UT : 1,		CONFIG : 'N U T, 0, 0, 0',
	X =  1125.569  mm,	Y =   539.568  mm,	Z =  1195.939  mm,
	W =   -37.197 deg,	P =    -5.451 deg,	R =   -16.720 deg
   GP2:
	UF : 1, UT : 1,
	J1=    90.000 deg,	J2=   100.000 deg
};
P[409]{
   GP1:
	UF : 1, UT : 1,		CONFIG : 'N U T, 0, 0, 0',
	X =  2172.569  mm,	Y =    47.854  mm,	Z =   147.939  mm,
	W =   -33.684 deg,	P =   -17.646 deg,	R =   -34.041 deg
   GP2:
	UF : 1, UT : 1,
	J1=    90.000 deg,	J2=   100.000 deg
};
P[410]{
   GP1:
	UF : 1, UT : 1,		CONFIG : 'N U T, 0, 0, 0',
	X =  2497.569  mm,	Y =    47.854  mm,	Z =   147.939  mm,
	W =   -33.684 deg,	P =   -17.646 deg,	R =   -34.041 deg
   GP2:
	UF : 1, UT : 1,
	J1=    90.000 deg,	J2=   100.000 deg
};
P[411]{
   GP1:
	UF : 1, UT : 1,		CONFIG : 'N U T, 0, 0, 0',
	X =  2519.938  mm,	Y =   -81.372  mm,	Z =   -32.158  mm,
	W =   -31.368 deg,	P =   -16.422 deg,	R =   -28.761 deg
   GP2:
	UF : 1, UT : 1,
	J1=    90.000 deg,	J2=   100.000 deg
};
P[412]{
   GP1:
	UF : 1, UT : 1,		CONFIG : 'N U T, 0, 0, 0',
	X =  2482.458  mm,	Y =   -80.069  mm,	Z =   -28.898  mm,
	W =   -25.037 deg,	P =   -25.315 deg,	R =   -46.367 deg
   GP2:
	UF : 1, UT : 1,
	J1=    90.000 deg,	J2=   100.000 deg
};
P[413]{
   GP1:
	UF : 1, UT : 1,		CONFIG : 'N U T, 0, 0, 0',
	X =  2453.629  mm,	Y =   -82.007  mm,	Z =   -26.243  mm,
	W =   -25.039 deg,	P =   -25.325 deg,	R =   -79.891 deg
   GP2:
	UF : 1, UT : 1,
	J1=    90.000 deg,	J2=   100.000 deg
};
P[414]{
   GP1:
	UF : 1, UT : 1,		CONFIG : 'N U T, 0, 0, 0',
	X =  2564.729  mm,	Y =    37.568  mm,	Z =   126.466  mm,
	W =   -31.566 deg,	P =   -16.651 deg,	R =   -48.456 deg
   GP2:
	UF : 1, UT : 1,
	J1=    90.000 deg,	J2=   100.000 deg
};
P[415]{
   GP1:
	UF : 1, UT : 1,		CONFIG : 'N U T, 0, 0, 0',
	X =  2361.283  mm,	Y =    58.394  mm,	Z =   147.939  mm,
	W =   -33.684 deg,	P =   -17.646 deg,	R =   -34.041 deg
   GP2:
	UF : 1, UT : 1,
	J1=    90.000 deg,	J2=   100.000 deg
};
P[416]{
   GP1:
	UF : 1, UT : 1,		CONFIG : 'N U T, 0, 0, 0',
	X =  2351.765  mm,	Y =   -85.833  mm,	Z =   -33.800  mm,
	W =   -31.948 deg,	P =   -15.141 deg,	R =   -17.031 deg
   GP2:
	UF : 1, UT : 1,
	J1=    90.000 deg,	J2=   100.000 deg
};
P[417]{
   GP1:
	UF : 1, UT : 1,		CONFIG : 'N U T, 0, 0, 0',
	X =  2394.846  mm,	Y =   -83.445  mm,	Z =   -32.390  mm,
	W =   -31.930 deg,	P =   -15.141 deg,	R =   -17.037 deg
   GP2:
	UF : 1, UT : 1,
	J1=    90.000 deg,	J2=   100.000 deg
};
P[418]{
   GP1:
	UF : 1, UT : 1,		CONFIG : 'N U T, 0, 0, 0',
	X =  2420.835  mm,	Y =   -83.306  mm,	Z =   -29.423  mm,
	W =   -24.232 deg,	P =   -24.716 deg,	R =   -17.035 deg
   GP2:
	UF : 1, UT : 1,
	J1=    90.000 deg,	J2=   100.000 deg
};
P[419]{
   GP1:
	UF : 1, UT : 1,		CONFIG : 'N U T, 0, 0, 0',
	X =  2371.614  mm,	Y =   -31.308  mm,	Z =    73.274  mm,
	W =   -26.718 deg,	P =   -22.770 deg,	R =   -10.639 deg
   GP2:
	UF : 1, UT : 1,
	J1=    90.000 deg,	J2=   100.000 deg
};
P[420]{
   GP1:
	UF : 1, UT : 1,		CONFIG : 'N U T, 0, 0, 0',
	X =  1125.569  mm,	Y =   539.568  mm,	Z =  1045.939  mm,
	W =   -37.197 deg,	P =    -5.451 deg,	R =   -16.720 deg
   GP2:
	UF : 1, UT : 1,
	J1=    90.000 deg,	J2=   100.000 deg
};
P[421]{
   GP1:
	UF : 1, UT : 1,		CONFIG : 'N U T, 0, 0, 0',
	X =  1125.569  mm,	Y =   539.568  mm,	Z =  1045.939  mm,
	W =      .249 deg,	P =    55.227 deg,	R =  -177.147 deg
   GP2:
	UF : 1, UT : 1,
	J1=    90.000 deg,	J2=    90.000 deg
};
P[422]{
   GP1:
	UF : 1, UT : 1,		CONFIG : 'N U T, 0, 0, -1',
	X =  2117.778  mm,	Y =   173.525  mm,	Z =  1006.395  mm,
	W =     -.647 deg,	P =    55.219 deg,	R =   156.602 deg
   GP2:
	UF : 1, UT : 1,
	J1=    90.000 deg,	J2=    90.000 deg
};
P[423]{
   GP1:
	UF : 1, UT : 1,		CONFIG : 'N U T, 0, 0, -1',
	X =  2129.658  mm,	Y =   151.797  mm,	Z =   832.903  mm,
	W =     2.981 deg,	P =    35.499 deg,	R =   160.128 deg
   GP2:
	UF : 1, UT : 1,
	J1=    90.000 deg,	J2=    90.000 deg
};
P[424]{
   GP1:
	UF : 1, UT : 1,		CONFIG : 'N U T, 0, 0, -1',
	X =  2137.350  mm,	Y =   177.465  mm,	Z =   833.508  mm,
	W =     2.985 deg,	P =    35.513 deg,	R =   160.120 deg
   GP2:
	UF : 1, UT : 1,
	J1=    90.000 deg,	J2=    90.000 deg
};
P[425]{
   GP1:
	UF : 1, UT : 1,		CONFIG : 'N U T, 0, 0, 0',
	X =  2130.020  mm,	Y =   199.847  mm,	Z =   830.984  mm,
	W =     2.986 deg,	P =    35.518 deg,	R =  -100.169 deg
   GP2:
	UF : 1, UT : 1,
	J1=    90.000 deg,	J2=    90.000 deg
};
P[426]{
   GP1:
	UF : 1, UT : 1,		CONFIG : 'N U T, 0, 0, 0',
	X =  2102.832  mm,	Y =   191.069  mm,	Z =   829.130  mm,
	W =     2.988 deg,	P =    35.514 deg,	R =   -13.075 deg
   GP2:
	UF : 1, UT : 1,
	J1=    90.000 deg,	J2=    90.000 deg
};
P[427]{
   GP1:
	UF : 1, UT : 1,		CONFIG : 'N U T, 0, 0, 0',
	X =  2088.170  mm,	Y =   149.785  mm,	Z =   828.888  mm,
	W =     2.984 deg,	P =    35.513 deg,	R =   -13.072 deg
   GP2:
	UF : 1, UT : 1,
	J1=    90.000 deg,	J2=    90.000 deg
};
P[428]{
   GP1:
	UF : 1, UT : 1,		CONFIG : 'N U T, 0, 0, 0',
	X =  2102.574  mm,	Y =   126.514  mm,	Z =   830.669  mm,
	W =     2.985 deg,	P =    35.513 deg,	R =    80.476 deg
   GP2:
	UF : 1, UT : 1,
	J1=    90.000 deg,	J2=    90.000 deg
};
P[429]{
   GP1:
	UF : 1, UT : 1,		CONFIG : 'N U T, 0, 0, 0',
	X =  2126.850  mm,	Y =   136.271  mm,	Z =   831.455  mm,
	W =     2.984 deg,	P =    35.513 deg,	R =   159.523 deg
   GP2:
	UF : 1, UT : 1,
	J1=    90.000 deg,	J2=    90.000 deg
};
P[430]{
   GP1:
	UF : 1, UT : 1,		CONFIG : 'N U T, 0, 0, 0',
	X =  2131.899  mm,	Y =   151.648  mm,	Z =   831.455  mm,
	W =     2.984 deg,	P =    35.513 deg,	R =   159.523 deg
   GP2:
	UF : 1, UT : 1,
	J1=    90.000 deg,	J2=    90.000 deg
};
P[431]{
   GP1:
	UF : 1, UT : 1,		CONFIG : 'N U T, 0, 0, 0',
	X =  2068.875  mm,	Y =   196.174  mm,	Z =   979.978  mm,
	W =      .815 deg,	P =    36.667 deg,	R =   159.784 deg
   GP2:
	UF : 1, UT : 1,
	J1=    90.000 deg,	J2=    90.000 deg
};
P[432]{
   GP1:
	UF : 1, UT : 1,		CONFIG : 'N U T, 0, 0, 0',
	X =  2127.874  mm,	Y =   249.175  mm,	Z =   979.977  mm,
	W =    -8.588 deg,	P =    43.492 deg,	R =    86.611 deg
   GP2:
	UF : 1, UT : 1,
	J1=    90.000 deg,	J2=    90.000 deg
};
P[433]{
   GP1:
	UF : 1, UT : 1,		CONFIG : 'N U T, 0, 0, 0',
	X =  2112.924  mm,	Y =   226.875  mm,	Z =   829.785  mm,
	W =    -2.360 deg,	P =    42.843 deg,	R =    86.536 deg
   GP2:
	UF : 1, UT : 1,
	J1=    90.000 deg,	J2=    90.000 deg
};
P[434]{
   GP1:
	UF : 1, UT : 1,		CONFIG : 'N U T, 0, 0, 0',
	X =  2202.613  mm,	Y =   227.153  mm,	Z =   829.824  mm,
	W =    -2.356 deg,	P =    42.846 deg,	R =    86.538 deg
   GP2:
	UF : 1, UT : 1,
	J1=    90.000 deg,	J2=    90.000 deg
};
P[435]{
   GP1:
	UF : 1, UT : 1,		CONFIG : 'N U T, 0, 0, 0',
	X =  2215.661  mm,	Y =   222.377  mm,	Z =   830.815  mm,
	W =    -2.493 deg,	P =    44.293 deg,	R =    56.655 deg
   GP2:
	UF : 1, UT : 1,
	J1=    90.000 deg,	J2=    90.000 deg
};
P[436]{
   GP1:
	UF : 1, UT : 1,		CONFIG : 'N U T, 0, 0, 0',
	X =  2222.874  mm,	Y =   213.385  mm,	Z =   828.313  mm,
	W =      .032 deg,	P =    44.143 deg,	R =    40.390 deg
   GP2:
	UF : 1, UT : 1,
	J1=    90.000 deg,	J2=    90.000 deg
};
P[437]{
   GP1:
	UF : 1, UT : 1,		CONFIG : 'N U T, 0, 0, 0',
	X =  2449.009  mm,	Y =   -44.468  mm,	Z =   827.867  mm,
	W =     -.128 deg,	P =    43.814 deg,	R =    45.335 deg
   GP2:
	UF : 1, UT : 1,
	J1=    90.000 deg,	J2=    90.000 deg
};
P[438]{
   GP1:
	UF : 1, UT : 1,		CONFIG : 'N U T, 0, 0, 0',
	X =  2454.781  mm,	Y =   -47.719  mm,	Z =   829.593  mm,
	W =      .165 deg,	P =    43.853 deg,	R =    54.355 deg
   GP2:
	UF : 1, UT : 1,
	J1=    90.000 deg,	J2=    90.000 deg
};
P[439]{
   GP1:
	UF : 1, UT : 1,		CONFIG : 'N U T, 0, 0, 0',
	X =  2459.541  mm,	Y =   -51.626  mm,	Z =   829.104  mm,
	W =    -1.320 deg,	P =    42.586 deg,	R =    55.587 deg
   GP2:
	UF : 1, UT : 1,
	J1=    90.000 deg,	J2=    90.000 deg
};
P[440]{
   GP1:
	UF : 1, UT : 1,		CONFIG : 'N U T, 0, 0, 0',
	X =  2655.978  mm,	Y =  -198.403  mm,	Z =   829.994  mm,
	W =   -30.974 deg,	P =    27.490 deg,	R =    12.667 deg
   GP2:
	UF : 1, UT : 1,
	J1=    90.000 deg,	J2=    90.000 deg
};
P[441]{
   GP1:
	UF : 1, UT : 1,		CONFIG : 'N U T, 0, 0, 0',
	X =  2672.856  mm,	Y =  -207.422  mm,	Z =   831.831  mm,
	W =   -30.972 deg,	P =    27.486 deg,	R =    12.662 deg
   GP2:
	UF : 1, UT : 1,
	J1=    90.000 deg,	J2=    90.000 deg
};
P[442]{
   GP1:
	UF : 1, UT : 1,		CONFIG : 'N U T, 0, 0, 0',
	X =  2657.997  mm,	Y =  -144.176  mm,	Z =   981.534  mm,
	W =   -36.400 deg,	P =    28.534 deg,	R =    31.709 deg
   GP2:
	UF : 1, UT : 1,
	J1=    90.000 deg,	J2=    90.000 deg
};
P[443]{
   GP1:
	UF : 1, UT : 1,		CONFIG : 'N U T, 0, 0, 0',
	X =   997.713  mm,	Y =    11.153  mm,	Z =   981.534  mm,
	W =   -36.400 deg,	P =    28.534 deg,	R =    23.998 deg
   GP2:
	UF : 1, UT : 1,
	J1=    90.000 deg,	J2=    90.000 deg
};
P[444]{
   GP1:
	UF : 1, UT : 1,		CONFIG : 'N U T, 0, 0, 0',
	X =   997.713  mm,	Y =  -220.683  mm,	Z =   981.533  mm,
	W =   -43.636 deg,	P =   -12.296 deg,	R =    70.660 deg
   GP2:
	UF : 1, UT : 1,
	J1=    80.000 deg,	J2=    90.000 deg
};
P[445]{
   GP1:
	UF : 1, UT : 1,		CONFIG : 'N U T, 0, 0, 0',
	X =  2009.713  mm,	Y =  -220.683  mm,	Z =   311.533  mm,
	W =   -43.636 deg,	P =   -12.296 deg,	R =    70.660 deg
   GP2:
	UF : 1, UT : 1,
	J1=    80.000 deg,	J2=    90.000 deg
};
P[446]{
   GP1:
	UF : 1, UT : 1,		CONFIG : 'N U T, 0, 0, 0',
	X =  2033.303  mm,	Y =   -34.036  mm,	Z =   121.326  mm,
	W =   -38.665 deg,	P =    -2.420 deg,	R =   142.728 deg
   GP2:
	UF : 1, UT : 1,
	J1=    80.000 deg,	J2=    90.000 deg
};
P[447]{
   GP1:
	UF : 1, UT : 1,		CONFIG : 'N U T, 0, 0, 0',
	X =  2073.851  mm,	Y =    35.924  mm,	Z =    12.285  mm,
	W =   -30.951 deg,	P =    -2.135 deg,	R =   142.491 deg
   GP2:
	UF : 1, UT : 1,
	J1=    80.000 deg,	J2=    90.000 deg
};
P[448]{
   GP1:
	UF : 1, UT : 1,		CONFIG : 'N U T, 0, 0, 0',
	X =  2117.748  mm,	Y =    -4.566  mm,	Z =     3.630  mm,
	W =   -28.504 deg,	P =     6.349 deg,	R =   142.803 deg
   GP2:
	UF : 1, UT : 1,
	J1=    80.000 deg,	J2=    90.000 deg
};
P[449]{
   GP1:
	UF : 1, UT : 1,		CONFIG : 'N U T, 0, 0, 0',
	X =  2124.001  mm,	Y =   -12.191  mm,	Z =     2.432  mm,
	W =   -27.562 deg,	P =     5.114 deg,	R =   139.578 deg
   GP2:
	UF : 1, UT : 1,
	J1=    80.000 deg,	J2=    90.000 deg
};
P[450]{
   GP1:
	UF : 1, UT : 1,		CONFIG : 'N U T, 0, 0, 0',
	X =  2130.131  mm,	Y =   -20.247  mm,	Z =     1.791  mm,
	W =   -27.580 deg,	P =     5.122 deg,	R =   136.990 deg
   GP2:
	UF : 1, UT : 1,
	J1=    80.000 deg,	J2=    90.000 deg
};
P[451]{
   GP1:
	UF : 1, UT : 1,		CONFIG : 'N U T, 0, 0, 0',
	X =  2251.754  mm,	Y =  -187.747  mm,	Z =   -18.626  mm,
	W =   -36.464 deg,	P =    -8.806 deg,	R =   122.583 deg
   GP2:
	UF : 1, UT : 1,
	J1=    80.000 deg,	J2=    90.000 deg
};
P[452]{
   GP1:
	UF : 1, UT : 1,		CONFIG : 'N U T, 0, 0, 0',
	X =  2260.659  mm,	Y =  -197.463  mm,	Z =   -20.538  mm,
	W =   -36.554 deg,	P =   -11.684 deg,	R =   125.973 deg
   GP2:
	UF : 1, UT : 1,
	J1=    80.000 deg,	J2=    90.000 deg
};
P[453]{
   GP1:
	UF : 1, UT : 1,		CONFIG : 'N U T, 0, 0, 0',
	X =  2269.185  mm,	Y =  -206.886  mm,	Z =   -21.960  mm,
	W =   -36.304 deg,	P =   -14.510 deg,	R =   128.303 deg
   GP2:
	UF : 1, UT : 1,
	J1=    80.000 deg,	J2=    90.000 deg
};
P[454]{
   GP1:
	UF : 1, UT : 1,		CONFIG : 'N U T, 0, 0, 0',
	X =  2511.863  mm,	Y =  -435.567  mm,	Z =   -65.547  mm,
	W =   -23.381 deg,	P =   -31.779 deg,	R =    95.136 deg
   GP2:
	UF : 1, UT : 1,
	J1=    80.000 deg,	J2=    90.000 deg
};
P[455]{
   GP1:
	UF : 1, UT : 1,		CONFIG : 'N U T, 0, 0, 0',
	X =  2535.927  mm,	Y =  -449.078  mm,	Z =   -69.737  mm,
	W =   -18.431 deg,	P =   -37.735 deg,	R =   100.755 deg
   GP2:
	UF : 1, UT : 1,
	J1=    80.000 deg,	J2=    90.000 deg
};
P[456]{
   GP1:
	UF : 1, UT : 1,		CONFIG : 'N U T, 0, 0, 0',
	X =  2558.091  mm,	Y =  -453.543  mm,	Z =   -73.418  mm,
	W =   -18.771 deg,	P =   -39.987 deg,	R =   104.546 deg
   GP2:
	UF : 1, UT : 1,
	J1=    80.000 deg,	J2=    90.000 deg
};
P[457]{
   GP1:
	UF : 1, UT : 1,		CONFIG : 'N U T, 0, 0, 0',
	X =  2574.982  mm,	Y =  -457.797  mm,	Z =   -77.599  mm,
	W =   -22.267 deg,	P =   -37.927 deg,	R =   106.779 deg
   GP2:
	UF : 1, UT : 1,
	J1=    80.000 deg,	J2=    90.000 deg
};
P[458]{
   GP1:
	UF : 1, UT : 1,		CONFIG : 'N U T, 0, 0, 0',
	X =  2621.992  mm,	Y =  -529.847  mm,	Z =   -85.920  mm,
	W =   -33.012 deg,	P =   -16.164 deg,	R =    66.999 deg
   GP2:
	UF : 1, UT : 1,
	J1=    80.000 deg,	J2=    90.000 deg
};
P[459]{
   GP1:
	UF : 1, UT : 1,		CONFIG : 'N U T, 0, 0, 0',
	X =  2621.958  mm,	Y =  -548.775  mm,	Z =   -86.023  mm,
	W =   -33.009 deg,	P =   -16.162 deg,	R =    66.994 deg
   GP2:
	UF : 1, UT : 1,
	J1=    80.000 deg,	J2=    90.000 deg
};
P[460]{
   GP1:
	UF : 1, UT : 1,		CONFIG : 'N U T, 0, 0, 0',
	X =  2620.833  mm,	Y =  -724.953  mm,	Z =   -86.008  mm,
	W =   -27.674 deg,	P =   -22.322 deg,	R =    54.091 deg
   GP2:
	UF : 1, UT : 1,
	J1=    80.000 deg,	J2=    90.000 deg
};
P[461]{
   GP1:
	UF : 1, UT : 1,		CONFIG : 'N U T, 0, 0, 0',
	X =  2576.687  mm,	Y =  -716.670  mm,	Z =    -1.123  mm,
	W =   -27.687 deg,	P =   -22.321 deg,	R =    54.103 deg
   GP2:
	UF : 1, UT : 1,
	J1=    80.000 deg,	J2=    90.000 deg
};
P[462]{
   GP1:
	UF : 1, UT : 1,		CONFIG : 'N U T, 0, 0, 0',
	X =  2532.411  mm,	Y =  -819.670  mm,	Z =    -1.123  mm,
	W =   -27.687 deg,	P =   -22.321 deg,	R =    54.103 deg
   GP2:
	UF : 1, UT : 1,
	J1=    80.000 deg,	J2=    90.000 deg
};
P[463]{
   GP1:
	UF : 1, UT : 1,		CONFIG : 'N U T, 0, 0, 0',
	X =  2550.739  mm,	Y =  -832.902  mm,	Z =   -76.728  mm,
	W =   -27.690 deg,	P =   -22.316 deg,	R =    54.107 deg
   GP2:
	UF : 1, UT : 1,
	J1=    80.000 deg,	J2=    90.000 deg
};
P[464]{
   GP1:
	UF : 1, UT : 1,		CONFIG : 'N U T, 0, 0, 0',
	X =  2551.660  mm,	Y =  -813.166  mm,	Z =   -76.438  mm,
	W =   -27.682 deg,	P =   -22.308 deg,	R =    54.092 deg
   GP2:
	UF : 1, UT : 1,
	J1=    80.000 deg,	J2=    90.000 deg
};
P[465]{
   GP1:
	UF : 1, UT : 1,		CONFIG : 'N U T, 0, 0, 0',
	X =  2565.317  mm,	Y =  -801.232  mm,	Z =   -77.060  mm,
	W =   -27.686 deg,	P =   -22.321 deg,	R =    23.348 deg
   GP2:
	UF : 1, UT : 1,
	J1=    80.000 deg,	J2=    90.000 deg
};
P[466]{
   GP1:
	UF : 1, UT : 1,		CONFIG : 'N U T, 0, 0, 0',
	X =  2576.762  mm,	Y =  -796.353  mm,	Z =   -82.224  mm,
	W =   -33.350 deg,	P =   -11.305 deg,	R =    17.629 deg
   GP2:
	UF : 1, UT : 1,
	J1=    80.000 deg,	J2=    90.000 deg
};
P[467]{
   GP1:
	UF : 1, UT : 1,		CONFIG : 'N U T, 0, 0, 0',
	X =  2611.385  mm,	Y =  -766.607  mm,	Z =   -84.979  mm,
	W =   -30.071 deg,	P =    -4.704 deg,	R =    42.986 deg
   GP2:
	UF : 1, UT : 1,
	J1=    80.000 deg,	J2=    90.000 deg
};
P[468]{
   GP1:
	UF : 1, UT : 1,		CONFIG : 'N U T, 0, 0, 0',
	X =  2624.754  mm,	Y =  -718.507  mm,	Z =   -86.108  mm,
	W =   -25.591 deg,	P =   -24.735 deg,	R =    48.858 deg
   GP2:
	UF : 1, UT : 1,
	J1=    80.000 deg,	J2=    90.000 deg
};
P[469]{
   GP1:
	UF : 1, UT : 1,		CONFIG : 'N U T, 0, 0, 0',
	X =  2566.235  mm,	Y =  -721.088  mm,	Z =   115.103  mm,
	W =   -35.203 deg,	P =   -31.584 deg,	R =    53.410 deg
   GP2:
	UF : 1, UT : 1,
	J1=    80.000 deg,	J2=    90.000 deg
};
P[470]{
   GP1:
	UF : 1, UT : 1,		CONFIG : 'N U T, 0, 0, 0',
	X =  1323.235  mm,	Y =  -721.088  mm,	Z =   524.103  mm,
	W =   -35.203 deg,	P =   -31.584 deg,	R =    53.410 deg
   GP2:
	UF : 1, UT : 1,
	J1=    80.000 deg,	J2=    90.000 deg
};
P[471]{
   GP1:
	UF : 1, UT : 1,		CONFIG : 'N U T, 0, 0, 1',
	X =  1085.059  mm,	Y =   -93.088  mm,	Z =   524.103  mm,
	W =    -5.111 deg,	P =    43.836 deg,	R =   172.642 deg
   GP2:
	UF : 1, UT : 1,
	J1=    80.000 deg,	J2=    90.000 deg
};
P[472]{
   GP1:
	UF : 1, UT : 1,		CONFIG : 'N U T, 0, 0, 1',
	X =   916.718  mm,	Y =  -171.225  mm,	Z =  1504.038  mm,
	W =    97.453 deg,	P =    88.349 deg,	R =   -88.494 deg
   GP2:
	UF : 1, UT : 1,
	J1=    80.000 deg,	J2=    90.000 deg
};
P[473]{
   GP1:
	UF : 1, UT : 1,		CONFIG : 'N U T, 0, 0, 0',
	X =   922.816  mm,	Y =    -9.239  mm,	Z =  2168.306  mm,
	W =     -.010 deg,	P =   -45.000 deg,	R =     0.000 deg
   GP2:
	UF : 1, UT : 1,
	J1=    90.000 deg,	J2=   -90.000 deg
};
P[474]{
   GP1:
	UF : 1, UT : 1,		CONFIG : 'N U T, 0, 0, -1',
	X =  1499.817  mm,	Y = -1083.239  mm,	Z =   440.877  mm,
	W =   -44.578 deg,	P =    -6.914 deg,	R =    83.049 deg
   GP2:
	UF : 1, UT : 1,
	J1=    90.000 deg,	J2=   -90.000 deg
};
P[475]{
   GP1:
	UF : 1, UT : 1,		CONFIG : 'N U T, 0, 0, -1',
	X =  2355.816  mm,	Y =  -998.239  mm,	Z =    94.877  mm,
	W =   -44.578 deg,	P =    -6.914 deg,	R =    83.049 deg
   GP2:
	UF : 1, UT : 1,
	J1=    90.000 deg,	J2=   -90.000 deg
};
P[476]{
   GP1:
	UF : 1, UT : 1,		CONFIG : 'N U T, 0, 0, -1',
	X =  2380.661  mm,	Y =  -855.649  mm,	Z =   109.732  mm,
	W =   -44.580 deg,	P =    -6.907 deg,	R =    83.042 deg
   GP2:
	UF : 1, UT : 1,
	J1=    90.000 deg,	J2=   -90.000 deg
};
P[477]{
   GP1:
	UF : 1, UT : 1,		CONFIG : 'N U T, 0, 0, -1',
	X =  2494.854  mm,	Y =  -857.680  mm,	Z =    -8.806  mm,
	W =   -44.580 deg,	P =    -6.907 deg,	R =    84.735 deg
   GP2:
	UF : 1, UT : 1,
	J1=    90.000 deg,	J2=   -90.000 deg
};
P[478]{
   GP1:
	UF : 1, UT : 1,		CONFIG : 'N U T, 0, 0, -1',
	X =  2494.926  mm,	Y =  -777.781  mm,	Z =    -9.320  mm,
	W =   -44.580 deg,	P =    -6.907 deg,	R =    84.735 deg
   GP2:
	UF : 1, UT : 1,
	J1=    90.000 deg,	J2=   -90.000 deg
};
P[479]{
   GP1:
	UF : 1, UT : 1,		CONFIG : 'N U T, 0, 0, -1',
	X =  2373.746  mm,	Y =  -828.779  mm,	Z =   224.191  mm,
	W =   -44.579 deg,	P =    -6.907 deg,	R =   101.186 deg
   GP2:
	UF : 1, UT : 1,
	J1=    90.000 deg,	J2=   -90.000 deg
};
P[480]{
   GP1:
	UF : 1, UT : 1,		CONFIG : 'N U T, 0, 0, 0',
	X =  2376.848  mm,	Y =  -600.055  mm,	Z =   228.526  mm,
	W =   -47.568 deg,	P =      .065 deg,	R =    50.370 deg
   GP2:
	UF : 1, UT : 1,
	J1=    90.000 deg,	J2=   -90.000 deg
};
P[481]{
   GP1:
	UF : 1, UT : 1,		CONFIG : 'N U T, 0, 0, -1',
	X =  2443.747  mm,	Y =  -697.351  mm,	Z =    99.482  mm,
	W =   -41.825 deg,	P =    18.388 deg,	R =    51.054 deg
   GP2:
	UF : 1, UT : 1,
	J1=    90.000 deg,	J2=   -90.000 deg
};
P[482]{
   GP1:
	UF : 1, UT : 1,		CONFIG : 'N U T, 0, 0, 0',
	X =  2518.619  mm,	Y =  -755.627  mm,	Z =    -6.486  mm,
	W =   -39.981 deg,	P =    14.824 deg,	R =    17.712 deg
   GP2:
	UF : 1, UT : 1,
	J1=    90.000 deg,	J2=   -90.000 deg
};
P[483]{
   GP1:
	UF : 1, UT : 1,		CONFIG : 'N U T, 0, 0, 0',
	X =  2567.877  mm,	Y =  -756.992  mm,	Z =    -7.047  mm,
	W =   -39.981 deg,	P =    14.824 deg,	R =    17.712 deg
   GP2:
	UF : 1, UT : 1,
	J1=    90.000 deg,	J2=   -90.000 deg
};
P[484]{
   GP1:
	UF : 1, UT : 1,		CONFIG : 'N U T, 0, 0, 0',
	X =  2443.747  mm,	Y =  -697.351  mm,	Z =    99.482  mm,
	W =   -41.825 deg,	P =    18.388 deg,	R =    51.054 deg
   GP2:
	UF : 1, UT : 1,
	J1=    90.000 deg,	J2=   -90.000 deg
};
P[485]{
   GP1:
	UF : 1, UT : 1,		CONFIG : 'N U T, 0, 0, 0',
	X =  2443.747  mm,	Y =  -697.351  mm,	Z =   245.196  mm,
	W =   -57.120 deg,	P =     5.483 deg,	R =    47.853 deg
   GP2:
	UF : 1, UT : 1,
	J1=    90.000 deg,	J2=   -90.000 deg
};
P[486]{
   GP1:
	UF : 1, UT : 1,		CONFIG : 'N U T, 0, 0, 0',
	X =  1415.176  mm,	Y =  -697.351  mm,	Z =   245.196  mm,
	W =   -57.120 deg,	P =     5.483 deg,	R =    47.853 deg
   GP2:
	UF : 1, UT : 1,
	J1=    90.000 deg,	J2=   -90.000 deg
};
P[487]{
   GP1:
	UF : 1, UT : 1,		CONFIG : 'N U T, 0, 0, 0',
	X =  1415.175  mm,	Y =  -361.351  mm,	Z =   492.217  mm,
	W =    -2.074 deg,	P =   -10.233 deg,	R =    32.173 deg
   GP2:
	UF : 1, UT : 1,
	J1=    90.000 deg,	J2=  -135.000 deg
};
P[488]{
   GP1:
	UF : 1, UT : 1,		CONFIG : 'N U T, 0, 0, 0',
	X =  2670.175  mm,	Y =  -174.351  mm,	Z =   333.217  mm,
	W =     1.417 deg,	P =   -10.343 deg,	R =    12.808 deg
   GP2:
	UF : 1, UT : 1,
	J1=    90.000 deg,	J2=  -135.000 deg
};
P[489]{
   GP1:
	UF : 1, UT : 1,		CONFIG : 'N U T, 0, 0, 0',
	X =  2752.964  mm,	Y =  -168.876  mm,	Z =   176.244  mm,
	W =    -1.647 deg,	P =    -7.143 deg,	R =    13.032 deg
   GP2:
	UF : 1, UT : 1,
	J1=    90.000 deg,	J2=  -135.000 deg
};
P[490]{
   GP1:
	UF : 1, UT : 1,		CONFIG : 'N U T, 0, 0, 0',
	X =  2865.942  mm,	Y =  -168.094  mm,	Z =   177.218  mm,
	W =    -5.450 deg,	P =   -22.504 deg,	R =    14.017 deg
   GP2:
	UF : 1, UT : 1,
	J1=    90.000 deg,	J2=  -135.000 deg
};
P[491]{
   GP1:
	UF : 1, UT : 1,		CONFIG : 'N U T, 0, 0, 0',
	X =  2838.021  mm,	Y =  -168.157  mm,	Z =   249.822  mm,
	W =    -7.346 deg,	P =   -29.104 deg,	R =    14.845 deg
   GP2:
	UF : 1, UT : 1,
	J1=    90.000 deg,	J2=  -135.000 deg
};
P[492]{
   GP1:
	UF : 1, UT : 1,		CONFIG : 'N U T, 0, 0, 0',
	X =  2372.538  mm,	Y =  -278.569  mm,	Z =   249.822  mm,
	W =    -1.017 deg,	P =    -4.421 deg,	R =    12.975 deg
   GP2:
	UF : 1, UT : 1,
	J1=    90.000 deg,	J2=  -135.000 deg
};
P[493]{
   GP1:
	UF : 1, UT : 1,		CONFIG : 'N U T, 0, 0, 0',
	X =  2379.984  mm,	Y =  -271.988  mm,	Z =    87.998  mm,
	W =      .003 deg,	P =      .001 deg,	R =    -2.945 deg
   GP2:
	UF : 1, UT : 1,
	J1=    90.000 deg,	J2=  -135.000 deg
};
P[494]{
   GP1:
	UF : 1, UT : 1,		CONFIG : 'N U T, 0, 0, 0',
	X =  2755.499  mm,	Y =  -271.313  mm,	Z =    89.477  mm,
	W =      .076 deg,	P =    -1.495 deg,	R =    -2.941 deg
   GP2:
	UF : 1, UT : 1,
	J1=    90.000 deg,	J2=  -135.000 deg
};
P[495]{
   GP1:
	UF : 1, UT : 1,		CONFIG : 'N U T, 0, 0, 0',
	X =  2656.405  mm,	Y =  -272.702  mm,	Z =   254.628  mm,
	W =     0.000 deg,	P =    -6.880 deg,	R =    -2.940 deg
   GP2:
	UF : 1, UT : 1,
	J1=    90.000 deg,	J2=  -135.000 deg
};
P[496]{
   GP1:
	UF : 1, UT : 1,		CONFIG : 'N U T, 0, 0, 0',
	X =  2489.404  mm,	Y =   -49.702  mm,	Z =    81.225  mm,
	W =    43.945 deg,	P =   -11.174 deg,	R =     1.639 deg
   GP2:
	UF : 1, UT : 1,
	J1=    90.000 deg,	J2=   -90.000 deg
};
P[497]{
   GP1:
	UF : 1, UT : 1,		CONFIG : 'N U T, 0, 0, 0',
	X =  2489.404  mm,	Y =    82.676  mm,	Z =    70.893  mm,
	W =    39.708 deg,	P =   -23.339 deg,	R =    15.773 deg
   GP2:
	UF : 1, UT : 1,
	J1=    90.000 deg,	J2=   -90.000 deg
};
P[498]{
   GP1:
	UF : 1, UT : 1,		CONFIG : 'N U T, 0, 0, 0',
	X =  2504.732  mm,	Y =   163.801  mm,	Z =    -7.840  mm,
	W =    37.870 deg,	P =   -26.386 deg,	R =    31.563 deg
   GP2:
	UF : 1, UT : 1,
	J1=    90.000 deg,	J2=   -90.000 deg
};
P[499]{
   GP1:
	UF : 1, UT : 1,		CONFIG : 'N U T, 0, 0, 0',
	X =  2464.249  mm,	Y =   164.384  mm,	Z =    -7.847  mm,
	W =    37.874 deg,	P =   -26.389 deg,	R =    31.563 deg
   GP2:
	UF : 1, UT : 1,
	J1=    90.000 deg,	J2=   -90.000 deg
};
P[500]{
   GP1:
	UF : 1, UT : 1,		CONFIG : 'N U T, 0, 0, 0',
	X =  2444.114  mm,	Y =   163.873  mm,	Z =    -8.034  mm,
	W =    40.554 deg,	P =   -21.460 deg,	R =    53.231 deg
   GP2:
	UF : 1, UT : 1,
	J1=    90.000 deg,	J2=   -90.000 deg
};
P[501]{
   GP1:
	UF : 1, UT : 1,		CONFIG : 'N U T, 0, 0, 0',
	X =  2489.404  mm,	Y =    82.676  mm,	Z =    70.893  mm,
	W =    42.059 deg,	P =   -17.938 deg,	R =    23.331 deg
   GP2:
	UF : 1, UT : 1,
	J1=    90.000 deg,	J2=   -90.000 deg
};
P[502]{
   GP1:
	UF : 1, UT : 1,		CONFIG : 'N U T, 0, 0, 0',
	X =  2489.404  mm,	Y =  -188.988  mm,	Z =    81.225  mm,
	W =    43.034 deg,	P =    14.904 deg,	R =   -25.132 deg
   GP2:
	UF : 1, UT : 1,
	J1=    90.000 deg,	J2=   -90.000 deg
};
P[503]{
   GP1:
	UF : 1, UT : 1,		CONFIG : 'N U T, 0, 0, 0',
	X =  1670.833  mm,	Y =  -188.988  mm,	Z =    81.225  mm,
	W =    43.034 deg,	P =    14.904 deg,	R =   -25.132 deg
   GP2:
	UF : 1, UT : 1,
	J1=    90.000 deg,	J2=   -90.000 deg
};
P[504]{
   GP1:
	UF : 1, UT : 1,		CONFIG : 'N U T, 0, 0, 0',
	X =  1685.665  mm,	Y =   -64.872  mm,	Z =   -18.365  mm,
	W =    41.394 deg,	P =    19.519 deg,	R =   -17.046 deg
   GP2:
	UF : 1, UT : 1,
	J1=    90.000 deg,	J2=   -90.000 deg
};
P[505]{
   GP1:
	UF : 1, UT : 1,		CONFIG : 'N U T, 0, 0, 0',
	X =  1655.518  mm,	Y =   -66.180  mm,	Z =   -18.364  mm,
	W =    41.393 deg,	P =    19.514 deg,	R =   -16.107 deg
   GP2:
	UF : 1, UT : 1,
	J1=    90.000 deg,	J2=   -90.000 deg
};
P[506]{
   GP1:
	UF : 1, UT : 1,		CONFIG : 'N U T, 0, 0, 0',
	X =  1644.071  mm,	Y =   -64.443  mm,	Z =   -18.488  mm,
	W =    41.392 deg,	P =    19.514 deg,	R =     3.473 deg
   GP2:
	UF : 1, UT : 1,
	J1=    90.000 deg,	J2=   -90.000 deg
};
P[507]{
   GP1:
	UF : 1, UT : 1,		CONFIG : 'N U T, 0, 0, 0',
	X =  1635.702  mm,	Y =   -66.864  mm,	Z =   -17.244  mm,
	W =    41.392 deg,	P =    19.514 deg,	R =    24.112 deg
   GP2:
	UF : 1, UT : 1,
	J1=    90.000 deg,	J2=   -90.000 deg
};
P[508]{
   GP1:
	UF : 1, UT : 1,		CONFIG : 'N U T, 0, 0, 0',
	X =  1608.120  mm,	Y =   -97.236  mm,	Z =   -17.308  mm,
	W =    37.029 deg,	P =    27.659 deg,	R =    15.298 deg
   GP2:
	UF : 1, UT : 1,
	J1=    90.000 deg,	J2=   -90.000 deg
};
P[509]{
   GP1:
	UF : 1, UT : 1,		CONFIG : 'N U T, 0, 0, 0',
	X =  1588.118  mm,	Y =  -108.567  mm,	Z =   -16.888  mm,
	W =    38.940 deg,	P =    23.604 deg,	R =   -29.723 deg
   GP2:
	UF : 1, UT : 1,
	J1=    90.000 deg,	J2=   -90.000 deg
};
P[510]{
   GP1:
	UF : 1, UT : 1,		CONFIG : 'N U T, 0, 0, 0',
	X =  1562.037  mm,	Y =   -85.294  mm,	Z =   -16.902  mm,
	W =    36.730 deg,	P =    28.082 deg,	R =  -109.081 deg
   GP2:
	UF : 1, UT : 1,
	J1=    90.000 deg,	J2=   -90.000 deg
};
P[511]{
   GP1:
	UF : 1, UT : 1,		CONFIG : 'N U T, 0, 0, 0',
	X =  1556.914  mm,	Y =   -40.647  mm,	Z =   -16.118  mm,
	W =    36.727 deg,	P =    28.082 deg,	R =  -114.509 deg
   GP2:
	UF : 1, UT : 1,
	J1=    90.000 deg,	J2=   -90.000 deg
};
P[512]{
   GP1:
	UF : 1, UT : 1,		CONFIG : 'N U T, 0, 0, 0',
	X =  1556.835  mm,	Y =   -36.070  mm,	Z =   -15.557  mm,
	W =    39.289 deg,	P =    28.081 deg,	R =   -80.638 deg
   GP2:
	UF : 1, UT : 1,
	J1=    90.000 deg,	J2=   -90.000 deg
};
P[513]{
   GP1:
	UF : 1, UT : 1,		CONFIG : 'N U T, 0, 0, 0',
	X =  1548.450  mm,	Y =   -29.796  mm,	Z =   -15.951  mm,
	W =    36.729 deg,	P =    28.085 deg,	R =   -43.976 deg
   GP2:
	UF : 1, UT : 1,
	J1=    90.000 deg,	J2=   -90.000 deg
};
P[514]{
   GP1:
	UF : 1, UT : 1,		CONFIG : 'N U T, 0, 0, 0',
	X =  1541.843  mm,	Y =   -26.526  mm,	Z =   -17.050  mm,
	W =    36.730 deg,	P =    28.085 deg,	R =   -43.977 deg
   GP2:
	UF : 1, UT : 1,
	J1=    90.000 deg,	J2=   -90.000 deg
};
P[515]{
   GP1:
	UF : 1, UT : 1,		CONFIG : 'N U T, 0, 0, 0',
	X =  1439.819  mm,	Y =  -288.523  mm,	Z =   263.807  mm,
	W =    40.466 deg,	P =    21.645 deg,	R =   -45.635 deg
   GP2:
	UF : 1, UT : 1,
	J1=    90.000 deg,	J2=   -90.000 deg
};
P[516]{
   GP1:
	UF : 1, UT : 1,		CONFIG : 'N U T, 0, 0, 0',
	X =  2349.342  mm,	Y =  -184.523  mm,	Z =   120.807  mm,
	W =    49.996 deg,	P =    12.253 deg,	R =   -42.841 deg
   GP2:
	UF : 1, UT : 1,
	J1=    90.000 deg,	J2=   -90.000 deg
};
P[517]{
   GP1:
	UF : 1, UT : 1,		CONFIG : 'N U T, 0, 0, 0',
	X =  2349.342  mm,	Y =    87.477  mm,	Z =   100.131  mm,
	W =    41.080 deg,	P =   -17.089 deg,	R =    29.592 deg
   GP2:
	UF : 1, UT : 1,
	J1=    90.000 deg,	J2=   -90.000 deg
};
P[518]{
   GP1:
	UF : 1, UT : 1,		CONFIG : 'N U T, 0, 0, 0',
	X =  2359.776  mm,	Y =   167.003  mm,	Z =    -8.816  mm,
	W =    38.121 deg,	P =   -25.966 deg,	R =    27.297 deg
   GP2:
	UF : 1, UT : 1,
	J1=    90.000 deg,	J2=   -90.000 deg
};
P[519]{
   GP1:
	UF : 1, UT : 1,		CONFIG : 'N U T, 0, 0, 0',
	X =  2406.274  mm,	Y =   166.697  mm,	Z =    -9.876  mm,
	W =    38.121 deg,	P =   -25.966 deg,	R =    27.297 deg
   GP2:
	UF : 1, UT : 1,
	J1=    90.000 deg,	J2=   -90.000 deg
};
P[520]{
   GP1:
	UF : 1, UT : 1,		CONFIG : 'N U T, 0, 0, 0',
	X =  2420.811  mm,	Y =   162.873  mm,	Z =    -7.347  mm,
	W =     9.855 deg,	P =   -38.956 deg,	R =    41.531 deg
   GP2:
	UF : 1, UT : 1,
	J1=    89.988 deg,	J2=   -90.001 deg
};
P[521]{
   GP1:
	UF : 1, UT : 1,		CONFIG : 'N U T, 0, 0, 0',
	X =  2355.377  mm,	Y =    87.835  mm,	Z =    47.968  mm,
	W =    34.887 deg,	P =   -26.988 deg,	R =    21.909 deg
   GP2:
	UF : 1, UT : 1,
	J1=    90.000 deg,	J2=   -90.000 deg
};
P[522]{
   GP1:
	UF : 1, UT : 1,		CONFIG : 'N U T, 0, 0, 0',
	X =  2349.342  mm,	Y =  -184.523  mm,	Z =   120.807  mm,
	W =    49.996 deg,	P =    12.253 deg,	R =   -42.841 deg
   GP2:
	UF : 1, UT : 1,
	J1=    90.000 deg,	J2=   -90.000 deg
};
P[523]{
   GP1:
	UF : 1, UT : 1,		CONFIG : 'N U T, 0, 0, 0',
	X =  1289.342  mm,	Y =  -184.523  mm,	Z =   120.807  mm,
	W =    49.996 deg,	P =    12.253 deg,	R =   -42.841 deg
   GP2:
	UF : 1, UT : 1,
	J1=    90.000 deg,	J2=   -90.000 deg
};
P[524]{
   GP1:
	UF : 1, UT : 1,		CONFIG : 'N U T, 0, 0, 0',
	X =  1152.199  mm,	Y =   223.477  mm,	Z =   120.807  mm,
	W =     5.452 deg,	P =    45.384 deg,	R =    96.559 deg
   GP2:
	UF : 1, UT : 1,
	J1=    90.000 deg,	J2=   -90.000 deg
};
P[525]{
   GP1:
	UF : 1, UT : 1,		CONFIG : 'N U T, 0, 0, 0',
	X =  1744.798  mm,	Y =   208.477  mm,	Z =    36.380  mm,
	W =   -35.057 deg,	P =    31.336 deg,	R =    18.229 deg
   GP2:
	UF : 1, UT : 1,
	J1=    90.000 deg,	J2=   -90.000 deg
};
P[526]{
   GP1:
	UF : 1, UT : 1,		CONFIG : 'N U T, 0, 0, 0',
	X =  1671.414  mm,	Y =   189.046  mm,	Z =   -15.712  mm,
	W =   -36.940 deg,	P =    22.774 deg,	R =   -15.979 deg
   GP2:
	UF : 1, UT : 1,
	J1=    90.000 deg,	J2=   -90.000 deg
};
P[527]{
   GP1:
	UF : 1, UT : 1,		CONFIG : 'N U T, 0, 0, 0',
	X =  1704.592  mm,	Y =   193.463  mm,	Z =   -14.287  mm,
	W =   -36.936 deg,	P =    22.774 deg,	R =    39.322 deg
   GP2:
	UF : 1, UT : 1,
	J1=    90.000 deg,	J2=   -90.000 deg
};
P[528]{
   GP1:
	UF : 1, UT : 1,		CONFIG : 'N U T, 0, 0, 0',
	X =  1976.573  mm,	Y =   191.971  mm,	Z =   -16.183  mm,
	W =   -36.940 deg,	P =    22.774 deg,	R =    39.323 deg
   GP2:
	UF : 1, UT : 1,
	J1=    90.000 deg,	J2=   -90.000 deg
};
P[529]{
   GP1:
	UF : 1, UT : 1,		CONFIG : 'N U T, 0, 0, 0',
	X =  1990.474  mm,	Y =   191.565  mm,	Z =   -18.105  mm,
	W =   -40.749 deg,	P =    13.396 deg,	R =    62.815 deg
   GP2:
	UF : 1, UT : 1,
	J1=    90.000 deg,	J2=   -90.000 deg
};
P[530]{
   GP1:
	UF : 1, UT : 1,		CONFIG : 'N U T, 0, 0, 0',
	X =  1983.329  mm,	Y =   227.532  mm,	Z =    32.278  mm,
	W =   -37.049 deg,	P =    22.562 deg,	R =    41.911 deg
   GP2:
	UF : 1, UT : 1,
	J1=    90.000 deg,	J2=   -90.000 deg
};
P[531]{
   GP1:
	UF : 1, UT : 1,		CONFIG : 'N U T, 0, 0, 0',
	X =  2295.778  mm,	Y =   288.199  mm,	Z =    71.302  mm,
	W =   -37.045 deg,	P =    22.566 deg,	R =    41.912 deg
   GP2:
	UF : 1, UT : 1,
	J1=    83.000 deg,	J2=   -90.000 deg
};
P[532]{
   GP1:
	UF : 1, UT : 1,		CONFIG : 'N U T, 0, 0, 0',
	X =  2506.193  mm,	Y =   208.629  mm,	Z =    36.065  mm,
	W =   -42.488 deg,	P =     1.840 deg,	R =   -59.515 deg
   GP2:
	UF : 1, UT : 1,
	J1=    83.000 deg,	J2=   -90.000 deg
};
P[533]{
   GP1:
	UF : 1, UT : 1,		CONFIG : 'N U T, 0, 0, 0',
	X =  2502.331  mm,	Y =   124.533  mm,	Z =    32.277  mm,
	W =   -42.488 deg,	P =     1.841 deg,	R =   -72.344 deg
   GP2:
	UF : 1, UT : 1,
	J1=    83.000 deg,	J2=   -90.000 deg
};
P[534]{
   GP1:
	UF : 1, UT : 1,		CONFIG : 'N U T, 0, 0, 0',
	X =  2392.053  mm,	Y =    84.549  mm,	Z =   -21.907  mm,
	W =   -47.015 deg,	P =     6.660 deg,	R =   -51.412 deg
   GP2:
	UF : 1, UT : 1,
	J1=    83.000 deg,	J2=   -90.000 deg
};
P[535]{
   GP1:
	UF : 1, UT : 1,		CONFIG : 'N U T, 0, 0, 0',
	X =  2391.109  mm,	Y =   106.727  mm,	Z =   -21.577  mm,
	W =   -47.008 deg,	P =     6.653 deg,	R =   -83.994 deg
   GP2:
	UF : 1, UT : 1,
	J1=    83.000 deg,	J2=   -90.000 deg
};
P[536]{
   GP1:
	UF : 1, UT : 1,		CONFIG : 'N U T, 0, 0, 0',
	X =  2390.648  mm,	Y =   140.871  mm,	Z =   -20.910  mm,
	W =   -47.989 deg,	P =     7.881 deg,	R =   -87.078 deg
   GP2:
	UF : 1, UT : 1,
	J1=    83.000 deg,	J2=   -90.000 deg
};
P[537]{
   GP1:
	UF : 1, UT : 1,		CONFIG : 'N U T, 0, 0, 0',
	X =  2393.525  mm,	Y =   163.570  mm,	Z =   -20.785  mm,
	W =   -47.988 deg,	P =     7.880 deg,	R =  -106.126 deg
   GP2:
	UF : 1, UT : 1,
	J1=    83.000 deg,	J2=   -90.000 deg
};
P[538]{
   GP1:
	UF : 1, UT : 1,		CONFIG : 'N U T, 0, 0, 0',
	X =  2502.331  mm,	Y =   124.533  mm,	Z =    32.277  mm,
	W =   -42.488 deg,	P =     1.841 deg,	R =   -72.344 deg
   GP2:
	UF : 1, UT : 1,
	J1=    83.000 deg,	J2=   -90.000 deg
};
P[539]{
   GP1:
	UF : 1, UT : 1,		CONFIG : 'N U T, 0, 0, 0',
	X =  2502.330  mm,	Y =   227.533  mm,	Z =    32.277  mm,
	W =   -46.494 deg,	P =   -14.946 deg,	R =     1.465 deg
   GP2:
	UF : 1, UT : 1,
	J1=    83.000 deg,	J2=   -90.000 deg
};
P[540]{
   GP1:
	UF : 1, UT : 1,		CONFIG : 'N U T, 0, 0, 0',
	X =  2378.330  mm,	Y =   227.532  mm,	Z =    38.468  mm,
	W =   -46.494 deg,	P =   -14.946 deg,	R =     1.465 deg
   GP2:
	UF : 1, UT : 1,
	J1=    90.000 deg,	J2=   -90.000 deg
};
P[541]{
   GP1:
	UF : 1, UT : 1,		CONFIG : 'N U T, 0, 0, 0',
	X =  2366.142  mm,	Y =   180.100  mm,	Z =    -9.199  mm,
	W =   -44.813 deg,	P =    -4.559 deg,	R =    -2.484 deg
   GP2:
	UF : 1, UT : 1,
	J1=    90.000 deg,	J2=   -90.000 deg
};
P[542]{
   GP1:
	UF : 1, UT : 1,		CONFIG : 'N U T, 0, 0, 0',
	X =  2505.035  mm,	Y =   180.287  mm,	Z =    -9.109  mm,
	W =   -44.818 deg,	P =    -4.562 deg,	R =    -2.490 deg
   GP2:
	UF : 1, UT : 1,
	J1=    90.000 deg,	J2=   -90.000 deg
};
P[543]{
   GP1:
	UF : 1, UT : 1,		CONFIG : 'N U T, 0, 0, 0',
	X =  2497.995  mm,	Y =   234.683  mm,	Z =    53.964  mm,
	W =   -44.990 deg,	P =    -1.038 deg,	R =    17.559 deg
   GP2:
	UF : 1, UT : 1,
	J1=    90.000 deg,	J2=   -90.000 deg
};
P[544]{
   GP1:
	UF : 1, UT : 1,		CONFIG : 'N U T, 0, 0, 0',
	X =  2294.995  mm,	Y =   234.683  mm,	Z =    53.964  mm,
	W =   -44.990 deg,	P =    -1.038 deg,	R =    17.559 deg
   GP2:
	UF : 1, UT : 1,
	J1=    90.000 deg,	J2=   -90.000 deg
};
P[545]{
   GP1:
	UF : 1, UT : 1,		CONFIG : 'N U T, 0, 0, 0',
	X =  2294.995  mm,	Y =   134.683  mm,	Z =    53.965  mm,
	W =   -44.990 deg,	P =    -1.038 deg,	R =    17.559 deg
   GP2:
	UF : 1, UT : 1,
	J1=    90.000 deg,	J2=   -90.000 deg
};
P[546]{
   GP1:
	UF : 1, UT : 1,		CONFIG : 'N U T, 0, 0, 0',
	X =  2363.074  mm,	Y =    82.607  mm,	Z =    -8.621  mm,
	W =   -44.379 deg,	P =     8.160 deg,	R =    14.035 deg
   GP2:
	UF : 1, UT : 1,
	J1=    90.000 deg,	J2=   -90.000 deg
};
P[547]{
   GP1:
	UF : 1, UT : 1,		CONFIG : 'N U T, 0, 0, 0',
	X =  2414.311  mm,	Y =    81.629  mm,	Z =    -8.521  mm,
	W =   -44.393 deg,	P =     8.163 deg,	R =    14.043 deg
   GP2:
	UF : 1, UT : 1,
	J1=    90.000 deg,	J2=   -90.000 deg
};
P[548]{
   GP1:
	UF : 1, UT : 1,		CONFIG : 'N U T, 0, 0, 0',
	X =  2420.856  mm,	Y =    84.559  mm,	Z =    -6.348  mm,
	W =   -44.535 deg,	P =    -7.128 deg,	R =    33.228 deg
   GP2:
	UF : 1, UT : 1,
	J1=    90.000 deg,	J2=   -90.000 deg
};
P[549]{
   GP1:
	UF : 1, UT : 1,		CONFIG : 'N U T, 0, 0, 0',
	X =  2294.995  mm,	Y =   210.290  mm,	Z =    96.252  mm,
	W =   -44.990 deg,	P =    -1.038 deg,	R =    25.270 deg
   GP2:
	UF : 1, UT : 1,
	J1=    90.000 deg,	J2=   -90.000 deg
};
P[550]{
   GP1:
	UF : 1, UT : 1,		CONFIG : 'N U T, 0, 0, 0',
	X =  1218.995  mm,	Y =   210.290  mm,	Z =    96.253  mm,
	W =   -44.990 deg,	P =    -1.038 deg,	R =    25.270 deg
   GP2:
	UF : 1, UT : 1,
	J1=    90.000 deg,	J2=   -90.000 deg
};
P[551]{
   GP1:
	UF : 1, UT : 1,		CONFIG : 'N U T, 0, 0, 0',
	X =  1218.995  mm,	Y =  -175.710  mm,	Z =  1113.253  mm,
	W =   -44.990 deg,	P =    -1.038 deg,	R =    25.270 deg
   GP2:
	UF : 1, UT : 1,
	J1=    90.000 deg,	J2=   -90.000 deg
};
P[552]{
   GP1:
	UF : 1, UT : 1,		CONFIG : 'N U T, 0, 0, 0',
	X =  2322.394  mm,	Y =   -54.093  mm,	Z =   961.517  mm,
	W =    42.919 deg,	P =     3.331 deg,	R =   -15.173 deg
   GP2:
	UF : 1, UT : 1,
	J1=    90.000 deg,	J2=   -90.000 deg
};
P[553]{
   GP1:
	UF : 1, UT : 1,		CONFIG : 'N U T, 0, 0, 0',
	X =  2347.090  mm,	Y =    54.696  mm,	Z =   840.157  mm,
	W =    45.388 deg,	P =    17.262 deg,	R =    -1.525 deg
   GP2:
	UF : 1, UT : 1,
	J1=    90.000 deg,	J2=   -90.000 deg
};
P[554]{
   GP1:
	UF : 1, UT : 1,		CONFIG : 'N U T, 0, 0, 0',
	X =  2407.727  mm,	Y =    84.771  mm,	Z =   840.157  mm,
	W =    45.388 deg,	P =    17.262 deg,	R =    -1.525 deg
   GP2:
	UF : 1, UT : 1,
	J1=    90.000 deg,	J2=   -90.000 deg
};
P[555]{
   GP1:
	UF : 1, UT : 1,		CONFIG : 'N U T, 0, 0, 0',
	X =  2424.460  mm,	Y =    34.399  mm,	Z =   891.750  mm,
	W =    45.388 deg,	P =    17.262 deg,	R =    -1.525 deg
   GP2:
	UF : 1, UT : 1,
	J1=    90.000 deg,	J2=   -90.000 deg
};
P[556]{
   GP1:
	UF : 1, UT : 1,		CONFIG : 'N U T, 0, 0, 0',
	X =  2461.841  mm,	Y =   116.924  mm,	Z =   905.997  mm,
	W =     1.448 deg,	P =    40.366 deg,	R =    26.776 deg
   GP2:
	UF : 1, UT : 1,
	J1=    90.000 deg,	J2=   -90.000 deg
};
P[557]{
   GP1:
	UF : 1, UT : 1,		CONFIG : 'N U T, 0, 0, 0',
	X =  2411.910  mm,	Y =    90.376  mm,	Z =   839.563  mm,
	W =     1.454 deg,	P =    40.369 deg,	R =    26.792 deg
   GP2:
	UF : 1, UT : 1,
	J1=    90.000 deg,	J2=   -90.000 deg
};
P[558]{
   GP1:
	UF : 1, UT : 1,		CONFIG : 'N U T, 0, 0, 0',
	X =  2400.458  mm,	Y =   114.292  mm,	Z =   839.623  mm,
	W =     1.448 deg,	P =    40.366 deg,	R =    26.776 deg
   GP2:
	UF : 1, UT : 1,
	J1=    90.000 deg,	J2=   -90.000 deg
};
P[559]{
   GP1:
	UF : 1, UT : 1,		CONFIG : 'N U T, 0, 0, 0',
	X =  2448.220  mm,	Y =   138.001  mm,	Z =   901.971  mm,
	W =     1.448 deg,	P =    40.366 deg,	R =    26.776 deg
   GP2:
	UF : 1, UT : 1,
	J1=    90.000 deg,	J2=   -90.000 deg
};
P[560]{
   GP1:
	UF : 1, UT : 1,		CONFIG : 'N U T, 0, 0, 0',
	X =  2256.717  mm,	Y =   -37.123  mm,	Z =  1005.877  mm,
	W =   -39.479 deg,	P =   -19.708 deg,	R =    39.669 deg
   GP2:
	UF : 1, UT : 1,
	J1=    90.000 deg,	J2=   -90.000 deg
};
P[561]{
   GP1:
	UF : 1, UT : 1,		CONFIG : 'F U T, 0, 0, 0',
	X =  2265.316  mm,	Y =   124.768  mm,	Z =   903.052  mm,
	W =   -46.224 deg,	P =   -25.156 deg,	R =    34.043 deg
   GP2:
	UF : 1, UT : 1,
	J1=    90.000 deg,	J2=   -90.000 deg
};
P[562]{
   GP1:
	UF : 1, UT : 1,		CONFIG : 'F U T, 0, 0, 0',
	X =  2330.795  mm,	Y =    79.737  mm,	Z =   841.199  mm,
	W =   -46.224 deg,	P =   -25.156 deg,	R =    34.043 deg
   GP2:
	UF : 1, UT : 1,
	J1=    90.000 deg,	J2=   -90.000 deg
};
P[563]{
   GP1:
	UF : 1, UT : 1,		CONFIG : 'F U T, 0, 0, 0',
	X =  2394.366  mm,	Y =   112.525  mm,	Z =   840.958  mm,
	W =   -46.224 deg,	P =   -25.155 deg,	R =    34.042 deg
   GP2:
	UF : 1, UT : 1,
	J1=    90.000 deg,	J2=   -90.000 deg
};
P[564]{
   GP1:
	UF : 1, UT : 1,		CONFIG : 'N U T, 0, 0, 0',
	X =  2189.899  mm,	Y =   169.121  mm,	Z =   881.852  mm,
	W =   -41.492 deg,	P =   -19.813 deg,	R =    37.650 deg
   GP2:
	UF : 1, UT : 1,
	J1=    90.000 deg,	J2=   -90.000 deg
};
P[565]{
   GP1:
	UF : 1, UT : 1,		CONFIG : 'N U T, 0, 0, 0',
	X =  2189.900  mm,	Y =   -28.744  mm,	Z =   939.390  mm,
	W =   -41.493 deg,	P =   -19.814 deg,	R =    37.650 deg
   GP2:
	UF : 1, UT : 1,
	J1=    90.000 deg,	J2=   -90.000 deg
};
P[566]{
   GP1:
	UF : 1, UT : 1,		CONFIG : 'N U T, 0, 0, 0',
	X =  1709.995  mm,	Y =  -228.567  mm,	Z =  1372.538  mm,
	W =    -4.515 deg,	P =      .965 deg,	R =    -2.729 deg
   GP2:
	UF : 1, UT : 1,
	J1=    90.000 deg,	J2=   -90.000 deg
};
P[567]{
   GP1:
	UF : 1, UT : 1,		CONFIG : 'N U T, 0, 0, 0',
	X =   922.816  mm,	Y =    -9.239  mm,	Z =  2168.306  mm,
	W =     -.010 deg,	P =   -45.000 deg,	R =     0.000 deg
   GP2:
	UF : 1, UT : 1,
	J1=    90.000 deg,	J2=  -100.000 deg
};
P[568]{
   GP1:
	UF : 1, UT : 1,		CONFIG : 'N U T, 0, 0, 0',
	X =  1001.816  mm,	Y =  -769.240  mm,	Z =   839.808  mm,
	W =     4.407 deg,	P =   -18.981 deg,	R =   -17.214 deg
   GP2:
	UF : 1, UT : 1,
	J1=    90.000 deg,	J2=  -100.000 deg
};
P[569]{
   GP1:
	UF : 1, UT : 1,		CONFIG : 'N U T, 0, 0, 0',
	X =  2120.817  mm,	Y =  -186.240  mm,	Z =   155.808  mm,
	W =    -4.184 deg,	P =     7.592 deg,	R =    43.674 deg
   GP2:
	UF : 1, UT : 1,
	J1=    90.000 deg,	J2=  -100.000 deg
};
P[570]{
   GP1:
	UF : 1, UT : 1,		CONFIG : 'N U T, 0, 0, 0',
	X =  2120.816  mm,	Y =   -28.525  mm,	Z =   155.808  mm,
	W =     2.218 deg,	P =    14.051 deg,	R =    70.281 deg
   GP2:
	UF : 1, UT : 1,
	J1=    90.000 deg,	J2=  -100.000 deg
};
P[571]{
   GP1:
	UF : 1, UT : 1,		CONFIG : 'N U T, 0, 0, 0',
	X =  2010.656  mm,	Y =   -98.489  mm,	Z =    -6.723  mm,
	W =    40.376 deg,	P =    23.931 deg,	R =    74.346 deg
   GP2:
	UF : 1, UT : 1,
	J1=    90.000 deg,	J2=  -100.000 deg
};
P[572]{
   GP1:
	UF : 1, UT : 1,		CONFIG : 'N U T, 0, 0, 0',
	X =  2009.129  mm,	Y =   124.302  mm,	Z =   -44.627  mm,
	W =    45.687 deg,	P =     4.511 deg,	R =    78.829 deg
   GP2:
	UF : 1, UT : 1,
	J1=    90.000 deg,	J2=  -100.000 deg
};
P[573]{
   GP1:
	UF : 1, UT : 1,		CONFIG : 'N U T, 0, 0, 0',
	X =  2120.816  mm,	Y =   -28.525  mm,	Z =   155.807  mm,
	W =     2.218 deg,	P =    14.051 deg,	R =    70.281 deg
   GP2:
	UF : 1, UT : 1,
	J1=    90.000 deg,	J2=  -100.000 deg
};
P[574]{
   GP1:
	UF : 1, UT : 1,		CONFIG : 'N U T, 0, 0, 0',
	X =  2120.817  mm,	Y =  -186.240  mm,	Z =   155.808  mm,
	W =    -4.184 deg,	P =     7.592 deg,	R =    43.674 deg
   GP2:
	UF : 1, UT : 1,
	J1=    90.000 deg,	J2=  -100.000 deg
};
P[575]{
   GP1:
	UF : 1, UT : 1,		CONFIG : 'N U T, 0, 0, 0',
	X =  2169.234  mm,	Y =  -186.240  mm,	Z =   155.807  mm,
	W =    28.994 deg,	P =   -15.433 deg,	R =    30.441 deg
   GP2:
	UF : 1, UT : 1,
	J1=    90.000 deg,	J2=   -90.000 deg
};
P[576]{
   GP1:
	UF : 1, UT : 1,		CONFIG : 'N U T, 0, 0, 0',
	X =  2230.271  mm,	Y =   -64.539  mm,	Z =    -1.822  mm,
	W =    44.892 deg,	P =    -3.427 deg,	R =     3.436 deg
   GP2:
	UF : 1, UT : 1,
	J1=    90.000 deg,	J2=   -90.000 deg
};
P[577]{
   GP1:
	UF : 1, UT : 1,		CONFIG : 'N U T, 0, 0, 0',
	X =  2260.320  mm,	Y =   -63.687  mm,	Z =    -1.783  mm,
	W =    44.897 deg,	P =    -3.424 deg,	R =     3.430 deg
   GP2:
	UF : 1, UT : 1,
	J1=    90.000 deg,	J2=   -90.000 deg
};
P[578]{
   GP1:
	UF : 1, UT : 1,		CONFIG : 'N U T, 0, 0, 0',
	X =  2171.101  mm,	Y =  -106.848  mm,	Z =    40.010  mm,
	W =    44.885 deg,	P =     3.628 deg,	R =    -3.635 deg
   GP2:
	UF : 1, UT : 1,
	J1=    90.000 deg,	J2=   -90.000 deg
};
P[579]{
   GP1:
	UF : 1, UT : 1,		CONFIG : 'N U T, 0, 0, 0',
	X =  2134.875  mm,	Y =   -62.293  mm,	Z =   -12.089  mm,
	W =    44.886 deg,	P =     3.630 deg,	R =    -4.912 deg
   GP2:
	UF : 1, UT : 1,
	J1=    90.000 deg,	J2=   -90.000 deg
};
P[580]{
   GP1:
	UF : 1, UT : 1,		CONFIG : 'N U T, 0, 0, 0',
	X =  2205.171  mm,	Y =   -64.816  mm,	Z =   -10.170  mm,
	W =    44.886 deg,	P =     3.630 deg,	R =    -4.912 deg
   GP2:
	UF : 1, UT : 1,
	J1=    90.000 deg,	J2=   -90.000 deg
};
P[581]{
   GP1:
	UF : 1, UT : 1,		CONFIG : 'N U T, 0, 0, 0',
	X =  2212.120  mm,	Y =   -62.897  mm,	Z =   -10.890  mm,
	W =    44.886 deg,	P =     3.630 deg,	R =   -11.550 deg
   GP2:
	UF : 1, UT : 1,
	J1=    90.000 deg,	J2=   -90.000 deg
};
P[582]{
   GP1:
	UF : 1, UT : 1,		CONFIG : 'N U T, 0, 0, 0',
	X =  2072.771  mm,	Y =  -106.847  mm,	Z =    40.010  mm,
	W =    44.885 deg,	P =     3.628 deg,	R =    -3.635 deg
   GP2:
	UF : 1, UT : 1,
	J1=    90.000 deg,	J2=   -90.000 deg
};
P[583]{
   GP1:
	UF : 1, UT : 1,		CONFIG : 'N U T, 0, 0, 0',
	X =  1984.534  mm,	Y =   -65.727  mm,	Z =   -17.955  mm,
	W =    44.885 deg,	P =     3.628 deg,	R =    -8.844 deg
   GP2:
	UF : 1, UT : 1,
	J1=    90.000 deg,	J2=   -90.000 deg
};
P[584]{
   GP1:
	UF : 1, UT : 1,		CONFIG : 'N U T, 0, 0, 0',
	X =  2097.268  mm,	Y =   -65.065  mm,	Z =   -17.473  mm,
	W =    44.885 deg,	P =     3.628 deg,	R =    -8.844 deg
   GP2:
	UF : 1, UT : 1,
	J1=    90.000 deg,	J2=   -90.000 deg
};
P[585]{
   GP1:
	UF : 1, UT : 1,		CONFIG : 'N U T, 0, 0, 0',
	X =  2112.828  mm,	Y =   -64.584  mm,	Z =   -16.753  mm,
	W =    41.205 deg,	P =   -19.972 deg,	R =    -8.013 deg
   GP2:
	UF : 1, UT : 1,
	J1=    90.000 deg,	J2=   -90.000 deg
};
P[586]{
   GP1:
	UF : 1, UT : 1,		CONFIG : 'N U T, 0, 0, 0',
	X =  1903.826  mm,	Y =  -198.100  mm,	Z =    98.030  mm,
	W =    40.690 deg,	P =   -21.162 deg,	R =    -6.795 deg
   GP2:
	UF : 1, UT : 1,
	J1=    90.000 deg,	J2=   -90.000 deg
};
P[587]{
   GP1:
	UF : 1, UT : 1,		CONFIG : 'N U T, 0, 0, 0',
	X =  1903.827  mm,	Y =  -198.100  mm,	Z =    98.030  mm,
	W =   -33.760 deg,	P =   -16.746 deg,	R =    41.760 deg
   GP2:
	UF : 1, UT : 1,
	J1=    90.000 deg,	J2=   -90.000 deg
};
P[588]{
   GP1:
	UF : 1, UT : 1,		CONFIG : 'N U T, 0, 0, 0',
	X =  2037.827  mm,	Y =  -117.100  mm,	Z =    98.030  mm,
	W =   -36.632 deg,	P =    -7.222 deg,	R =    55.482 deg
   GP2:
	UF : 1, UT : 1,
	J1=    90.000 deg,	J2=   -90.000 deg
};
P[589]{
   GP1:
	UF : 1, UT : 1,		CONFIG : 'N U T, 0, 0, 0',
	X =  2071.831  mm,	Y =  -111.826  mm,	Z =   -18.286  mm,
	W =   -37.503 deg,	P =      .971 deg,	R =    76.661 deg
   GP2:
	UF : 1, UT : 1,
	J1=    90.000 deg,	J2=   -90.000 deg
};
P[590]{
   GP1:
	UF : 1, UT : 1,		CONFIG : 'N U T, 0, 0, 0',
	X =  2101.801  mm,	Y =   -84.456  mm,	Z =   -18.286  mm,
	W =   -37.503 deg,	P =      .971 deg,	R =    85.242 deg
   GP2:
	UF : 1, UT : 1,
	J1=    90.000 deg,	J2=   -90.000 deg
};
P[591]{
   GP1:
	UF : 1, UT : 1,		CONFIG : 'N U T, 0, 0, 0',
	X =  2119.303  mm,	Y =   -69.097  mm,	Z =   -17.436  mm,
	W =   -37.503 deg,	P =      .971 deg,	R =   107.030 deg
   GP2:
	UF : 1, UT : 1,
	J1=    90.000 deg,	J2=   -90.000 deg
};
P[592]{
   GP1:
	UF : 1, UT : 1,		CONFIG : 'N U T, 0, 0, 0',
	X =  2055.659  mm,	Y =   -89.520  mm,	Z =    80.831  mm,
	W =   -33.519 deg,	P =   -11.367 deg,	R =    99.761 deg
   GP2:
	UF : 1, UT : 1,
	J1=    90.000 deg,	J2=   -90.000 deg
};
P[593]{
   GP1:
	UF : 1, UT : 1,		CONFIG : 'N U T, 0, 0, 1',
	X =  1095.659  mm,	Y =  -338.091  mm,	Z =    80.831  mm,
	W =   -14.565 deg,	P =    32.384 deg,	R =  -179.547 deg
   GP2:
	UF : 1, UT : 1,
	J1=    90.000 deg,	J2=   -90.000 deg
};
P[594]{
   GP1:
	UF : 1, UT : 1,		CONFIG : 'N U T, 0, 0, 1',
	X =  1464.711  mm,	Y =  -492.316  mm,	Z =  1452.110  mm,
	W =    59.113 deg,	P =    76.093 deg,	R =  -118.587 deg
   GP2:
	UF : 1, UT : 1,
	J1=    90.000 deg,	J2=   -90.000 deg
};
P[595]{
   GP1:
	UF : 1, UT : 1,		CONFIG : 'N U T, 0, 0, 1',
	X =  2120.659  mm,	Y =  -156.092  mm,	Z =   977.831  mm,
	W =    -2.744 deg,	P =    30.268 deg,	R =  -167.022 deg
   GP2:
	UF : 1, UT : 1,
	J1=    90.000 deg,	J2=   -90.000 deg
};
P[596]{
   GP1:
	UF : 1, UT : 1,		CONFIG : 'N U T, 0, 0, 1',
	X =  2129.923  mm,	Y =  -163.109  mm,	Z =   831.039  mm,
	W =     3.597 deg,	P =    39.858 deg,	R =  -158.843 deg
   GP2:
	UF : 1, UT : 1,
	J1=    90.000 deg,	J2=   -90.000 deg
};
P[597]{
   GP1:
	UF : 1, UT : 1,		CONFIG : 'N U T, 0, 0, 1',
	X =  2137.809  mm,	Y =  -186.248  mm,	Z =   831.044  mm,
	W =     2.770 deg,	P =    38.184 deg,	R =  -159.358 deg
   GP2:
	UF : 1, UT : 1,
	J1=    90.000 deg,	J2=   -90.000 deg
};
P[598]{
   GP1:
	UF : 1, UT : 1,		CONFIG : 'N U T, 0, 0, 0',
	X =  2125.992  mm,	Y =  -204.644  mm,	Z =   830.285  mm,
	W =     7.244 deg,	P =    45.395 deg,	R =   112.852 deg
   GP2:
	UF : 1, UT : 1,
	J1=    90.000 deg,	J2=   -90.000 deg
};
P[599]{
   GP1:
	UF : 1, UT : 1,		CONFIG : 'N U T, 0, 0, 0',
	X =  2100.015  mm,	Y =  -196.039  mm,	Z =   828.573  mm,
	W =     5.322 deg,	P =    47.573 deg,	R =    22.949 deg
   GP2:
	UF : 1, UT : 1,
	J1=    90.000 deg,	J2=   -90.000 deg
};
P[600]{
   GP1:
	UF : 1, UT : 1,		CONFIG : 'N U T, 0, 0, 0',
	X =  2086.616  mm,	Y =  -152.754  mm,	Z =   828.880  mm,
	W =      .306 deg,	P =    46.787 deg,	R =    19.130 deg
   GP2:
	UF : 1, UT : 1,
	J1=    90.000 deg,	J2=   -90.000 deg
};
P[601]{
   GP1:
	UF : 1, UT : 1,		CONFIG : 'N U T, 0, 0, 0',
	X =  2100.504  mm,	Y =  -134.531  mm,	Z =   832.401  mm,
	W =    -1.751 deg,	P =    45.025 deg,	R =   -76.985 deg
   GP2:
	UF : 1, UT : 1,
	J1=    90.000 deg,	J2=   -90.000 deg
};
P[602]{
   GP1:
	UF : 1, UT : 1,		CONFIG : 'N U T, 0, 0, 0',
	X =  2125.547  mm,	Y =  -142.237  mm,	Z =   829.698  mm,
	W =      .707 deg,	P =    41.168 deg,	R =  -163.588 deg
   GP2:
	UF : 1, UT : 1,
	J1=    90.000 deg,	J2=   -90.000 deg
};
P[603]{
   GP1:
	UF : 1, UT : 1,		CONFIG : 'N U T, 0, 0, 0',
	X =  2131.397  mm,	Y =  -162.602  mm,	Z =   829.829  mm,
	W =      .078 deg,	P =    40.942 deg,	R =  -164.204 deg
   GP2:
	UF : 1, UT : 1,
	J1=    90.000 deg,	J2=   -90.000 deg
};
P[604]{
   GP1:
	UF : 1, UT : 1,		CONFIG : 'N U T, 0, 0, 0',
	X =  2005.953  mm,	Y =  -131.336  mm,	Z =  1019.826  mm,
	W =    10.851 deg,	P =    41.306 deg,	R =  -172.082 deg
   GP2:
	UF : 1, UT : 1,
	J1=    90.000 deg,	J2=   -90.000 deg
};
P[605]{
   GP1:
	UF : 1, UT : 1,		CONFIG : 'N U T, 0, 0, 0',
	X =  2119.952  mm,	Y =  -275.231  mm,	Z =  1019.826  mm,
	W =     2.972 deg,	P =    30.278 deg,	R =   -91.159 deg
   GP2:
	UF : 1, UT : 1,
	J1=    90.000 deg,	J2=   -90.000 deg
};
P[606]{
   GP1:
	UF : 1, UT : 1,		CONFIG : 'N U T, 0, 0, 0',
	X =  2108.961  mm,	Y =  -235.302  mm,	Z =   830.555  mm,
	W =     -.443 deg,	P =    39.555 deg,	R =   -90.699 deg
   GP2:
	UF : 1, UT : 1,
	J1=    90.000 deg,	J2=   -90.000 deg
};
P[607]{
   GP1:
	UF : 1, UT : 1,		CONFIG : 'N U T, 0, 0, 0',
	X =  2201.336  mm,	Y =  -235.279  mm,	Z =   830.597  mm,
	W =     -.447 deg,	P =    39.555 deg,	R =   -90.703 deg
   GP2:
	UF : 1, UT : 1,
	J1=    90.000 deg,	J2=   -90.000 deg
};
P[608]{
   GP1:
	UF : 1, UT : 1,		CONFIG : 'N U T, 0, 0, 0',
	X =  2214.980  mm,	Y =  -233.048  mm,	Z =   831.869  mm,
	W =     -.447 deg,	P =    39.555 deg,	R =   -57.817 deg
   GP2:
	UF : 1, UT : 1,
	J1=    90.000 deg,	J2=   -90.000 deg
};
P[609]{
   GP1:
	UF : 1, UT : 1,		CONFIG : 'N U T, 0, 0, 0',
	X =  2222.918  mm,	Y =  -224.326  mm,	Z =   830.599  mm,
	W =     -.447 deg,	P =    39.555 deg,	R =   -44.058 deg
   GP2:
	UF : 1, UT : 1,
	J1=    90.000 deg,	J2=   -90.000 deg
};
P[610]{
   GP1:
	UF : 1, UT : 1,		CONFIG : 'N U T, 0, 0, 0',
	X =  2394.178  mm,	Y =   -28.001  mm,	Z =   831.741  mm,
	W =     -.034 deg,	P =    41.997 deg,	R =   -43.180 deg
   GP2:
	UF : 1, UT : 1,
	J1=    90.000 deg,	J2=   -90.000 deg
};
P[611]{
   GP1:
	UF : 1, UT : 1,		CONFIG : 'N U T, 0, 0, 0',
	X =  2450.792  mm,	Y =    35.777  mm,	Z =   832.312  mm,
	W =      .115 deg,	P =    42.764 deg,	R =   -49.054 deg
   GP2:
	UF : 1, UT : 1,
	J1=    90.000 deg,	J2=   -90.000 deg
};
P[612]{
   GP1:
	UF : 1, UT : 1,		CONFIG : 'N U T, 0, 0, 0',
	X =  2457.628  mm,	Y =    40.947  mm,	Z =   832.314  mm,
	W =      .115 deg,	P =    42.764 deg,	R =   -56.123 deg
   GP2:
	UF : 1, UT : 1,
	J1=    90.000 deg,	J2=   -90.000 deg
};
P[613]{
   GP1:
	UF : 1, UT : 1,		CONFIG : 'N U T, 0, 0, 0',
	X =  2521.514  mm,	Y =    87.672  mm,	Z =   832.133  mm,
	W =    11.971 deg,	P =    40.663 deg,	R =   -38.122 deg
   GP2:
	UF : 1, UT : 1,
	J1=    90.000 deg,	J2=   -90.000 deg
};
P[614]{
   GP1:
	UF : 1, UT : 1,		CONFIG : 'N U T, 0, 0, 0',
	X =  2650.676  mm,	Y =   184.582  mm,	Z =   832.304  mm,
	W =    27.597 deg,	P =    31.501 deg,	R =   -10.869 deg
   GP2:
	UF : 1, UT : 1,
	J1=    90.000 deg,	J2=   -90.000 deg
};
P[615]{
   GP1:
	UF : 1, UT : 1,		CONFIG : 'N U T, 0, 0, 0',
	X =  2693.013  mm,	Y =   190.209  mm,	Z =   894.682  mm,
	W =    28.386 deg,	P =    27.784 deg,	R =   -40.362 deg
   GP2:
	UF : 1, UT : 1,
	J1=    90.000 deg,	J2=   -90.000 deg
};
P[616]{
   GP1:
	UF : 1, UT : 1,		CONFIG : 'N U T, 0, 0, 0',
	X =   946.013  mm,	Y =   190.209  mm,	Z =   994.682  mm,
	W =    28.386 deg,	P =    27.784 deg,	R =   -40.362 deg
   GP2:
	UF : 1, UT : 1,
	J1=    90.000 deg,	J2=   -90.000 deg
};
P[617]{
   GP1:
	UF : 1, UT : 1,		CONFIG : 'N U T, 0, 0, 0',
	X =   946.013  mm,	Y =   190.209  mm,	Z =   326.110  mm,
	W =   -34.527 deg,	P =    19.136 deg,	R =    25.896 deg
   GP2:
	UF : 1, UT : 1,
	J1=    90.000 deg,	J2=   -90.000 deg
};
P[618]{
   GP1:
	UF : 1, UT : 1,		CONFIG : 'N U T, 0, 0, 0',
	X =  1715.261  mm,	Y =   113.066  mm,	Z =   168.110  mm,
	W =   -48.737 deg,	P =     8.784 deg,	R =     7.978 deg
   GP2:
	UF : 1, UT : 1,
	J1=    90.000 deg,	J2=   -90.000 deg
};
P[619]{
   GP1:
	UF : 1, UT : 1,		CONFIG : 'N U T, 0, 0, 0',
	X =  1959.340  mm,	Y =   -50.107  mm,	Z =    51.552  mm,
	W =   -51.898 deg,	P =     9.370 deg,	R =    14.305 deg
   GP2:
	UF : 1, UT : 1,
	J1=    90.000 deg,	J2=   -90.000 deg
};
P[620]{
   GP1:
	UF : 1, UT : 1,		CONFIG : 'N U T, 0, 0, 0',
	X =  1948.268  mm,	Y =   -49.653  mm,	Z =    51.537  mm,
	W =   -51.894 deg,	P =     9.366 deg,	R =     5.846 deg
   GP2:
	UF : 1, UT : 1,
	J1=    90.000 deg,	J2=   -90.000 deg
};
P[621]{
   GP1:
	UF : 1, UT : 1,		CONFIG : 'N U T, 0, 0, 0',
	X =  1696.243  mm,	Y =   -50.530  mm,	Z =    52.257  mm,
	W =   -51.894 deg,	P =     9.366 deg,	R =     5.846 deg
   GP2:
	UF : 1, UT : 1,
	J1=    90.000 deg,	J2=   -90.000 deg
};
P[622]{
   GP1:
	UF : 1, UT : 1,		CONFIG : 'N U T, 0, 0, 0',
	X =  1670.714  mm,	Y =   -48.833  mm,	Z =    54.913  mm,
	W =   -51.894 deg,	P =     9.366 deg,	R =   -32.596 deg
   GP2:
	UF : 1, UT : 1,
	J1=    90.000 deg,	J2=   -90.000 deg
};
P[623]{
   GP1:
	UF : 1, UT : 1,		CONFIG : 'N U T, 0, 0, 0',
	X =  1930.555  mm,	Y =    75.757  mm,	Z =   159.682  mm,
	W =   -51.903 deg,	P =     9.364 deg,	R =    21.482 deg
   GP2:
	UF : 1, UT : 1,
	J1=    90.000 deg,	J2=   -90.000 deg
};
P[624]{
   GP1:
	UF : 1, UT : 1,		CONFIG : 'N U T, 0, 0, 0',
	X =  2187.556  mm,	Y =    75.757  mm,	Z =   159.682  mm,
	W =   -51.227 deg,	P =   -13.564 deg,	R =     3.543 deg
   GP2:
	UF : 1, UT : 1,
	J1=    90.000 deg,	J2=   -90.000 deg
};
P[625]{
   GP1:
	UF : 1, UT : 1,		CONFIG : 'N U T, 0, 0, 0',
	X =  2224.519  mm,	Y =   -44.534  mm,	Z =    -1.819  mm,
	W =   -45.065 deg,	P =    -5.943 deg,	R =    -3.250 deg
   GP2:
	UF : 1, UT : 1,
	J1=    90.000 deg,	J2=   -90.000 deg
};
P[626]{
   GP1:
	UF : 1, UT : 1,		CONFIG : 'N U T, 0, 0, 0',
	X =  2262.967  mm,	Y =   -46.459  mm,	Z =    -2.708  mm,
	W =   -45.063 deg,	P =    -5.948 deg,	R =    -3.255 deg
   GP2:
	UF : 1, UT : 1,
	J1=    90.000 deg,	J2=   -90.000 deg
};
P[627]{
   GP1:
	UF : 1, UT : 1,		CONFIG : 'N U T, 0, 0, 0',
	X =  2185.536  mm,	Y =    -1.237  mm,	Z =    55.960  mm,
	W =   -44.735 deg,	P =    -5.491 deg,	R =    -5.516 deg
   GP2:
	UF : 1, UT : 1,
	J1=    90.000 deg,	J2=   -90.000 deg
};
P[628]{
   GP1:
	UF : 1, UT : 1,		CONFIG : 'N U T, 0, 0, 0',
	X =  2141.111  mm,	Y =   -46.149  mm,	Z =    -9.294  mm,
	W =   -44.730 deg,	P =    -5.491 deg,	R =    -5.523 deg
   GP2:
	UF : 1, UT : 1,
	J1=    90.000 deg,	J2=   -90.000 deg
};
P[629]{
   GP1:
	UF : 1, UT : 1,		CONFIG : 'N U T, 0, 0, 0',
	X =  2205.054  mm,	Y =   -46.149  mm,	Z =    -9.294  mm,
	W =   -44.730 deg,	P =    -5.491 deg,	R =    -5.523 deg
   GP2:
	UF : 1, UT : 1,
	J1=    90.000 deg,	J2=   -90.000 deg
};
P[630]{
   GP1:
	UF : 1, UT : 1,		CONFIG : 'N U T, 0, 0, 0',
	X =  2212.135  mm,	Y =   -45.578  mm,	Z =    -9.294  mm,
	W =   -44.730 deg,	P =    -5.491 deg,	R =    10.504 deg
   GP2:
	UF : 1, UT : 1,
	J1=    90.000 deg,	J2=   -90.000 deg
};
P[631]{
   GP1:
	UF : 1, UT : 1,		CONFIG : 'N U T, 0, 0, 0',
	X =  2095.621  mm,	Y =    -7.964  mm,	Z =    38.524  mm,
	W =   -44.735 deg,	P =    -5.491 deg,	R =    -5.516 deg
   GP2:
	UF : 1, UT : 1,
	J1=    90.000 deg,	J2=   -90.000 deg
};
P[632]{
   GP1:
	UF : 1, UT : 1,		CONFIG : 'N U T, 0, 0, 0',
	X =  2115.729  mm,	Y =   -45.526  mm,	Z =   -17.679  mm,
	W =   -44.735 deg,	P =    -5.490 deg,	R =    -5.517 deg
   GP2:
	UF : 1, UT : 1,
	J1=    90.000 deg,	J2=   -90.000 deg
};
P[633]{
   GP1:
	UF : 1, UT : 1,		CONFIG : 'N U T, 0, 0, 0',
	X =  2032.308  mm,	Y =   -46.092  mm,	Z =   -17.679  mm,
	W =   -44.735 deg,	P =    -5.490 deg,	R =    -5.517 deg
   GP2:
	UF : 1, UT : 1,
	J1=    90.000 deg,	J2=   -90.000 deg
};
P[634]{
   GP1:
	UF : 1, UT : 1,		CONFIG : 'N U T, 0, 0, 0',
	X =  2010.263  mm,	Y =   -47.292  mm,	Z =   -17.680  mm,
	W =   -44.735 deg,	P =    -5.490 deg,	R =   -41.540 deg
   GP2:
	UF : 1, UT : 1,
	J1=    90.000 deg,	J2=   -90.000 deg
};
P[635]{
   GP1:
	UF : 1, UT : 1,		CONFIG : 'N U T, 0, 0, 0',
	X =  2078.052  mm,	Y =    71.672  mm,	Z =   101.338  mm,
	W =   -44.734 deg,	P =    -5.490 deg,	R =     4.917 deg
   GP2:
	UF : 1, UT : 1,
	J1=    90.000 deg,	J2=   -90.000 deg
};
P[636]{
   GP1:
	UF : 1, UT : 1,		CONFIG : 'N U T, 0, 0, 0',
	X =  1302.053  mm,	Y =    71.672  mm,	Z =   101.339  mm,
	W =   -44.734 deg,	P =    -5.490 deg,	R =     4.917 deg
   GP2:
	UF : 1, UT : 1,
	J1=    90.000 deg,	J2=   -90.000 deg
};
P[637]{
   GP1:
	UF : 1, UT : 1,		CONFIG : 'N U T, 0, 0, 1',
	X =  1302.053  mm,	Y =    71.673  mm,	Z =   101.339  mm,
	W =    36.994 deg,	P =    27.707 deg,	R =  -122.588 deg
   GP2:
	UF : 1, UT : 1,
	J1=    90.000 deg,	J2=   -90.000 deg
};
P[638]{
   GP1:
	UF : 1, UT : 1,		CONFIG : 'N U T, 0, 0, 1',
	X =  1623.053  mm,	Y =   183.673  mm,	Z =    50.339  mm,
	W =    36.994 deg,	P =    27.707 deg,	R =  -122.588 deg
   GP2:
	UF : 1, UT : 1,
	J1=    90.000 deg,	J2=   -90.000 deg
};
P[639]{
   GP1:
	UF : 1, UT : 1,		CONFIG : 'N U T, 0, 0, 0',
	X =  1652.956  mm,	Y =   215.868  mm,	Z =   -13.936  mm,
	W =    34.857 deg,	P =    26.466 deg,	R =  -126.842 deg
   GP2:
	UF : 1, UT : 1,
	J1=    90.000 deg,	J2=   -90.000 deg
};
P[640]{
   GP1:
	UF : 1, UT : 1,		CONFIG : 'N U T, 0, 0, 1',
	X =  1654.227  mm,	Y =    -6.870  mm,	Z =   -18.681  mm,
	W =    36.965 deg,	P =    27.690 deg,	R =  -122.601 deg
   GP2:
	UF : 1, UT : 1,
	J1=    90.000 deg,	J2=   -90.000 deg
};
P[641]{
   GP1:
	UF : 1, UT : 1,		CONFIG : 'N U T, 0, 0, 0',
	X =  1654.396  mm,	Y =   -25.585  mm,	Z =   -18.765  mm,
	W =    37.080 deg,	P =    27.790 deg,	R =  -137.819 deg
   GP2:
	UF : 1, UT : 1,
	J1=    90.000 deg,	J2=   -90.000 deg
};
P[642]{
   GP1:
	UF : 1, UT : 1,		CONFIG : 'N U T, 0, 0, 0',
	X =  1532.379  mm,	Y =    48.074  mm,	Z =   132.806  mm,
	W =    36.993 deg,	P =    27.706 deg,	R =  -154.189 deg
   GP2:
	UF : 1, UT : 1,
	J1=    90.000 deg,	J2=   -90.000 deg
};
P[643]{
   GP1:
	UF : 1, UT : 1,		CONFIG : 'N U T, 0, 0, 0',
	X =  1491.379  mm,	Y =   161.074  mm,	Z =   377.806  mm,
	W =    23.939 deg,	P =    39.314 deg,	R =  -177.488 deg
   GP2:
	UF : 1, UT : 1,
	J1=    80.000 deg,	J2=   -90.000 deg
};
P[644]{
   GP1:
	UF : 1, UT : 1,		CONFIG : 'N U T, 0, 0, 0',
	X =  2049.380  mm,	Y =   161.074  mm,	Z =   177.806  mm,
	W =    23.939 deg,	P =    39.314 deg,	R =  -177.488 deg
   GP2:
	UF : 1, UT : 1,
	J1=    80.000 deg,	J2=   -90.000 deg
};
P[645]{
   GP1:
	UF : 1, UT : 1,		CONFIG : 'N U T, 0, 0, -1',
	X =  2049.380  mm,	Y =    -6.926  mm,	Z =   106.806  mm,
	W =    34.881 deg,	P =    30.459 deg,	R =  -142.693 deg
   GP2:
	UF : 1, UT : 1,
	J1=    80.000 deg,	J2=   -90.000 deg
};
P[646]{
   GP1:
	UF : 1, UT : 1,		CONFIG : 'N U T, 0, 0, 0',
	X =  2063.360  mm,	Y =   -46.552  mm,	Z =    14.408  mm,
	W =    27.118 deg,	P =    24.034 deg,	R =  -162.974 deg
   GP2:
	UF : 1, UT : 1,
	J1=    80.000 deg,	J2=   -90.000 deg
};
P[647]{
   GP1:
	UF : 1, UT : 1,		CONFIG : 'N U T, 0, 0, 1',
	X =  2070.201  mm,	Y =    -5.697  mm,	Z =    13.112  mm,
	W =    26.540 deg,	P =    23.909 deg,	R =  -139.397 deg
   GP2:
	UF : 0, UT : 1,
	J1=    80.000 deg,	J2=   -90.000 deg
};
P[648]{
   GP1:
	UF : 1, UT : 1,		CONFIG : 'N U T, 0, 0, 0',
	X =  2069.499  mm,	Y =    -1.522  mm,	Z =    13.452  mm,
	W =    26.543 deg,	P =    23.908 deg,	R =  -163.851 deg
   GP2:
	UF : 1, UT : 1,
	J1=    80.000 deg,	J2=   -90.000 deg
};
P[649]{
   GP1:
	UF : 1, UT : 1,		CONFIG : 'N U T, 0, 0, 0',
	X =  2079.957  mm,	Y =    14.618  mm,	Z =    14.062  mm,
	W =    17.949 deg,	P =    33.023 deg,	R =   153.341 deg
   GP2:
	UF : 1, UT : 1,
	J1=    80.000 deg,	J2=   -90.000 deg
};
P[650]{
   GP1:
	UF : 1, UT : 1,		CONFIG : 'N U T, 0, 0, 0',
	X =  2257.638  mm,	Y =   188.605  mm,	Z =   -17.721  mm,
	W =      .048 deg,	P =    36.127 deg,	R =   125.240 deg
   GP2:
	UF : 0, UT : 1,
	J1=    80.000 deg,	J2=   -90.000 deg
};
P[651]{
   GP1:
	UF : 1, UT : 1,		CONFIG : 'N U T, 0, 0, 0',
	X =  2269.957  mm,	Y =   197.647  mm,	Z =   -19.138  mm,
	W =     3.307 deg,	P =    33.871 deg,	R =   124.431 deg
   GP2:
	UF : 0, UT : 1,
	J1=    80.000 deg,	J2=   -90.000 deg
};
P[652]{
   GP1:
	UF : 1, UT : 1,		CONFIG : 'N U T, 0, 0, 0',
	X =  2281.172  mm,	Y =   204.541  mm,	Z =   -20.943  mm,
	W =     6.003 deg,	P =    35.927 deg,	R =   123.386 deg
   GP2:
	UF : 0, UT : 1,
	J1=    80.000 deg,	J2=   -90.000 deg
};
P[653]{
   GP1:
	UF : 1, UT : 1,		CONFIG : 'N U T, 0, 0, 0',
	X =  2386.760  mm,	Y =   271.261  mm,	Z =   -38.436  mm,
	W =     8.791 deg,	P =    37.202 deg,	R =   129.076 deg
   GP2:
	UF : 0, UT : 1,
	J1=    80.000 deg,	J2=   -90.000 deg
};
P[654]{
   GP1:
	UF : 1, UT : 1,		CONFIG : 'N U T, 0, 0, 0',
	X =  2402.059  mm,	Y =   281.172  mm,	Z =   -42.884  mm,
	W =    -2.502 deg,	P =    34.195 deg,	R =   123.652 deg
   GP2:
	UF : 0, UT : 1,
	J1=    80.000 deg,	J2=   -90.000 deg
};
P[655]{
   GP1:
	UF : 1, UT : 1,		CONFIG : 'N U T, 0, 0, 0',
	X =  2416.336  mm,	Y =   299.753  mm,	Z =   -44.208  mm,
	W =      .578 deg,	P =    31.078 deg,	R =   135.858 deg
   GP2:
	UF : 0, UT : 1,
	J1=    80.000 deg,	J2=   -90.000 deg
};
P[656]{
   GP1:
	UF : 1, UT : 1,		CONFIG : 'N U T, 0, 0, 0',
	X =  2499.975  mm,	Y =   418.494  mm,	Z =   -59.863  mm,
	W =   -18.687 deg,	P =    29.860 deg,	R =   100.231 deg
   GP2:
	UF : 0, UT : 1,
	J1=    80.000 deg,	J2=   -90.000 deg
};
P[657]{
   GP1:
	UF : 1, UT : 1,		CONFIG : 'N U T, 0, 0, 0',
	X =  2522.749  mm,	Y =   437.814  mm,	Z =   -61.500  mm,
	W =   -18.823 deg,	P =    32.557 deg,	R =    79.853 deg
   GP2:
	UF : 0, UT : 1,
	J1=    80.000 deg,	J2=   -90.000 deg
};
P[658]{
   GP1:
	UF : 1, UT : 1,		CONFIG : 'N U T, 0, 0, 0',
	X =  2555.836  mm,	Y =   446.395  mm,	Z =   -68.337  mm,
	W =   -16.509 deg,	P =    33.836 deg,	R =    74.966 deg
   GP2:
	UF : 0, UT : 1,
	J1=    80.000 deg,	J2=   -90.000 deg
};
P[659]{
   GP1:
	UF : 1, UT : 1,		CONFIG : 'N U T, 0, 0, 0',
	X =  2568.335  mm,	Y =   451.071  mm,	Z =   -68.337  mm,
	W =   -16.509 deg,	P =    33.836 deg,	R =    74.966 deg
   GP2:
	UF : 0, UT : 1,
	J1=    80.000 deg,	J2=   -90.000 deg
};
P[660]{
   GP1:
	UF : 1, UT : 1,		CONFIG : 'N U T, 0, 0, 0',
	X =  2604.215  mm,	Y =   477.246  mm,	Z =   -76.736  mm,
	W =   -17.687 deg,	P =    33.474 deg,	R =   110.394 deg
   GP2:
	UF : 0, UT : 1,
	J1=    80.000 deg,	J2=   -90.000 deg
};
P[661]{
   GP1:
	UF : 1, UT : 1,		CONFIG : 'N U T, 0, 0, 0',
	X =  2618.697  mm,	Y =   518.470  mm,	Z =   -81.888  mm,
	W =   -28.179 deg,	P =    11.270 deg,	R =   110.042 deg
   GP2:
	UF : 0, UT : 1,
	J1=    80.000 deg,	J2=   -90.000 deg
};
P[662]{
   GP1:
	UF : 1, UT : 1,		CONFIG : 'N U T, 0, 0, 0',
	X =  2619.516  mm,	Y =   709.528  mm,	Z =   -82.638  mm,
	W =   -28.920 deg,	P =    12.962 deg,	R =   109.018 deg
   GP2:
	UF : 0, UT : 1,
	J1=    80.000 deg,	J2=   -90.000 deg
};
P[663]{
   GP1:
	UF : 1, UT : 1,		CONFIG : 'N U T, 0, 0, 0',
	X =  2621.157  mm,	Y =   717.292  mm,	Z =   -84.163  mm,
	W =   -28.920 deg,	P =    12.962 deg,	R =    86.656 deg
   GP2:
	UF : 0, UT : 1,
	J1=    80.000 deg,	J2=   -90.000 deg
};
P[664]{
   GP1:
	UF : 1, UT : 1,		CONFIG : 'N U T, 0, 0, 0',
	X =  2623.715  mm,	Y =   724.341  mm,	Z =   -84.162  mm,
	W =   -28.920 deg,	P =    12.962 deg,	R =    81.288 deg
   GP2:
	UF : 0, UT : 1,
	J1=    80.000 deg,	J2=   -90.000 deg
};
P[665]{
   GP1:
	UF : 1, UT : 1,		CONFIG : 'N U T, 0, 0, 0',
	X =  2631.075  mm,	Y =   754.747  mm,	Z =   -85.027  mm,
	W =   -29.833 deg,	P =     9.276 deg,	R =    88.853 deg
   GP2:
	UF : 0, UT : 1,
	J1=    80.000 deg,	J2=   -90.000 deg
};
P[666]{
   GP1:
	UF : 1, UT : 1,		CONFIG : 'N U T, 0, 0, 0',
	X =  2630.091  mm,	Y =   766.127  mm,	Z =   -86.552  mm,
	W =   -33.769 deg,	P =      .741 deg,	R =   112.878 deg
   GP2:
	UF : 0, UT : 1,
	J1=    80.000 deg,	J2=   -90.000 deg
};
P[667]{
   GP1:
	UF : 1, UT : 1,		CONFIG : 'N U T, 0, 0, 0',
	X =  2507.109  mm,	Y =   731.136  mm,	Z =    16.168  mm,
	W =   -42.166 deg,	P =     5.515 deg,	R =   107.587 deg
   GP2:
	UF : 1, UT : 1,
	J1=    80.000 deg,	J2=   -90.000 deg
};
P[668]{
   GP1:
	UF : 1, UT : 1,		CONFIG : 'N U T, 0, 0, 0',
	X =  2507.109  mm,	Y =   801.136  mm,	Z =    16.168  mm,
	W =   -35.462 deg,	P =    25.069 deg,	R =   132.276 deg
   GP2:
	UF : 1, UT : 1,
	J1=    80.000 deg,	J2=   -90.000 deg
};
P[669]{
   GP1:
	UF : 1, UT : 1,		CONFIG : 'N U T, 0, 0, 0',
	X =  2547.891  mm,	Y =   822.808  mm,	Z =   -72.485  mm,
	W =   -31.199 deg,	P =     9.620 deg,	R =   105.426 deg
   GP2:
	UF : 1, UT : 1,
	J1=    80.000 deg,	J2=   -90.000 deg
};
P[670]{
   GP1:
	UF : 1, UT : 1,		CONFIG : 'N U T, 0, 0, 0',
	X =  2549.025  mm,	Y =   813.653  mm,	Z =   -72.568  mm,
	W =   -32.484 deg,	P =     1.246 deg,	R =    91.954 deg
   GP2:
	UF : 1, UT : 1,
	J1=    80.000 deg,	J2=   -90.000 deg
};
P[671]{
   GP1:
	UF : 1, UT : 1,		CONFIG : 'N U T, 0, 0, 0',
	X =  2556.443  mm,	Y =   796.316  mm,	Z =   -71.740  mm,
	W =   -29.311 deg,	P =   -14.722 deg,	R =   104.313 deg
   GP2:
	UF : 0, UT : 1,
	J1=    80.000 deg,	J2=   -90.000 deg
};
P[672]{
   GP1:
	UF : 1, UT : 1,		CONFIG : 'N U T, 0, 0, 0',
	X =  2576.844  mm,	Y =   790.013  mm,	Z =   -76.345  mm,
	W =    -3.324 deg,	P =   -34.459 deg,	R =   105.041 deg
   GP2:
	UF : 0, UT : 1,
	J1=    80.000 deg,	J2=   -90.000 deg
};
P[673]{
   GP1:
	UF : 1, UT : 1,		CONFIG : 'N U T, 0, 0, 0',
	X =  2600.397  mm,	Y =   789.960  mm,	Z =   -81.033  mm,
	W =    -3.272 deg,	P =   -34.453 deg,	R =   105.003 deg
   GP2:
	UF : 0, UT : 1,
	J1=    80.000 deg,	J2=   -90.000 deg
};
P[674]{
   GP1:
	UF : 1, UT : 1,		CONFIG : 'N U T, 0, 0, 0',
	X =  2617.219  mm,	Y =   781.118  mm,	Z =   -82.622  mm,
	W =     3.036 deg,	P =   -34.484 deg,	R =    65.941 deg
   GP2:
	UF : 1, UT : 1,
	J1=    80.000 deg,	J2=   -90.000 deg
};
P[675]{
   GP1:
	UF : 1, UT : 1,		CONFIG : 'N U T, 0, 0, 0',
	X =  2627.491  mm,	Y =   762.062  mm,	Z =   -83.870  mm,
	W =   -15.099 deg,	P =   -26.030 deg,	R =    67.737 deg
   GP2:
	UF : 0, UT : 1,
	J1=    80.000 deg,	J2=   -90.000 deg
};
P[676]{
   GP1:
	UF : 1, UT : 1,		CONFIG : 'N U T, 0, 0, 0',
	X =  2536.373  mm,	Y =   677.588  mm,	Z =   101.581  mm,
	W =   -11.653 deg,	P =   -32.812 deg,	R =    68.201 deg
   GP2:
	UF : 1, UT : 1,
	J1=    80.000 deg,	J2=   -90.000 deg
};
P[677]{
   GP1:
	UF : 1, UT : 1,		CONFIG : 'N U T, 0, 0, 1',
	X =  2379.054  mm,	Y =   340.913  mm,	Z =   218.031  mm,
	W =   -12.774 deg,	P =    75.193 deg,	R =  -178.717 deg
   GP2:
	UF : 1, UT : 1,
	J1=    80.000 deg,	J2=   -90.000 deg
};
P[678]{
   GP1:
	UF : 1, UT : 1,		CONFIG : 'N U T, 0, 0, 1',
	X =  1113.732  mm,	Y =   361.444  mm,	Z =   517.929  mm,
	W =    14.500 deg,	P =    75.040 deg,	R =  -140.487 deg
   GP2:
	UF : 1, UT : 1,
	J1=    80.000 deg,	J2=   -90.000 deg
};
P[679]{
   GP1:
	UF : 1, UT : 1,		CONFIG : 'N U T, 0, 0, 0',
	X =   922.816  mm,	Y =    -9.239  mm,	Z =  2168.306  mm,
	W =     -.010 deg,	P =   -45.000 deg,	R =     0.000 deg
   GP2:
	UF : 1, UT : 1,
	J1=   180.000 deg,	J2=  -150.000 deg
};
P[680]{
   GP1:
	UF : 1, UT : 1,		CONFIG : 'N U T, 0, 0, 0',
	X =   913.051  mm,	Y = -1107.917  mm,	Z =  1634.767  mm,
	W =    10.155 deg,	P =    42.864 deg,	R =  -126.216 deg
   GP2:
	UF : 1, UT : 1,
	J1=   180.000 deg,	J2=  -150.000 deg
};
P[681]{
   GP1:
	UF : 1, UT : 1,		CONFIG : 'N U T, 0, 0, 0',
	X =   813.817  mm,	Y = -1211.238  mm,	Z =  1026.306  mm,
	W =    24.190 deg,	P =   -39.178 deg,	R =    -6.255 deg
   GP2:
	UF : 1, UT : 1,
	J1=   180.000 deg,	J2=  -150.000 deg
};
P[682]{
   GP1:
	UF : 1, UT : 1,		CONFIG : 'N U T, 0, 0, 0',
	X =   968.817  mm,	Y = -1111.238  mm,	Z =   852.305  mm,
	W =    24.190 deg,	P =   -39.178 deg,	R =    -6.255 deg
   GP2:
	UF : 1, UT : 1,
	J1=   180.000 deg,	J2=  -150.000 deg
};
P[683]{
   GP1:
	UF : 1, UT : 1,		CONFIG : 'N U T, 0, 0, 0',
	X =  1053.046  mm,	Y = -1056.747  mm,	Z =   769.543  mm,
	W =    24.542 deg,	P =   -38.984 deg,	R =    -6.156 deg
   GP2:
	UF : 1, UT : 1,
	J1=   180.000 deg,	J2=  -150.000 deg
};
P[684]{
   GP1:
	UF : 1, UT : 1,		CONFIG : 'N U T, 0, 0, 0',
	X =  1094.890  mm,	Y = -1127.769  mm,	Z =   768.463  mm,
	W =    24.536 deg,	P =   -38.987 deg,	R =    -6.145 deg
   GP2:
	UF : 1, UT : 1,
	J1=   180.000 deg,	J2=  -150.000 deg
};
P[685]{
   GP1:
	UF : 1, UT : 1,		CONFIG : 'N U T, 0, 0, 0',
	X =   585.666  mm,	Y = -1195.897  mm,	Z =  1026.056  mm,
	W =    24.190 deg,	P =   -39.178 deg,	R =    -6.255 deg
   GP2:
	UF : 1, UT : 1,
	J1=   180.000 deg,	J2=  -150.000 deg
};
P[686]{
   GP1:
	UF : 1, UT : 1,		CONFIG : 'N U T, 0, 0, 0',
	X =   585.666  mm,	Y = -1195.897  mm,	Z =  1026.056  mm,
	W =   -11.844 deg,	P =    43.739 deg,	R =  -167.714 deg
   GP2:
	UF : 1, UT : 1,
	J1=   180.000 deg,	J2=  -150.000 deg
};
P[687]{
   GP1:
	UF : 1, UT : 1,		CONFIG : 'N U T, 0, 0, 0',
	X =   763.666  mm,	Y =  -662.897  mm,	Z =   826.056  mm,
	W =   -27.661 deg,	P =    37.026 deg,	R =   168.125 deg
   GP2:
	UF : 1, UT : 1,
	J1=   180.000 deg,	J2=  -150.000 deg
};
P[688]{
   GP1:
	UF : 1, UT : 1,		CONFIG : 'N U T, 0, 0, 0',
	X =   776.756  mm,	Y =  -578.766  mm,	Z =   774.376  mm,
	W =   -11.191 deg,	P =    42.605 deg,	R =  -165.904 deg
   GP2:
	UF : 1, UT : 1,
	J1=   180.000 deg,	J2=  -150.000 deg
};
P[689]{
   GP1:
	UF : 1, UT : 1,		CONFIG : 'N U T, 0, 0, 0',
	X =   923.650  mm,	Y =  -831.496  mm,	Z =   772.822  mm,
	W =     1.427 deg,	P =    43.776 deg,	R =  -152.542 deg
   GP2:
	UF : 1, UT : 1,
	J1=   180.000 deg,	J2=  -150.000 deg
};
P[690]{
   GP1:
	UF : 1, UT : 1,		CONFIG : 'N U T, 0, 0, 0',
	X =  1037.419  mm,	Y = -1025.988  mm,	Z =   770.961  mm,
	W =     -.115 deg,	P =    43.762 deg,	R =  -154.812 deg
   GP2:
	UF : 1, UT : 1,
	J1=   180.000 deg,	J2=  -150.000 deg
};
P[691]{
   GP1:
	UF : 1, UT : 1,		CONFIG : 'N U T, 0, 0, 0',
	X =   969.618  mm,	Y = -1090.804  mm,	Z =   854.949  mm,
	W =    41.435 deg,	P =    19.411 deg,	R =   -80.632 deg
   GP2:
	UF : 1, UT : 1,
	J1=   180.000 deg,	J2=  -150.000 deg
};
P[692]{
   GP1:
	UF : 1, UT : 1,		CONFIG : 'N U T, 0, 0, 0',
	X =   607.272  mm,	Y =  -642.803  mm,	Z =   854.949  mm,
	W =    44.809 deg,	P =     4.676 deg,	R =   -64.692 deg
   GP2:
	UF : 1, UT : 1,
	J1=   180.000 deg,	J2=  -150.000 deg
};
P[693]{
   GP1:
	UF : 1, UT : 1,		CONFIG : 'N U T, 0, 0, 0',
	X =   758.466  mm,	Y =  -545.960  mm,	Z =   772.606  mm,
	W =    33.386 deg,	P =   -31.996 deg,	R =   -21.225 deg
   GP2:
	UF : 1, UT : 1,
	J1=   180.000 deg,	J2=  -150.000 deg
};
P[694]{
   GP1:
	UF : 1, UT : 1,		CONFIG : 'N U T, 0, 0, 0',
	X =   710.278  mm,	Y =  -477.960  mm,	Z =   772.606  mm,
	W =    33.386 deg,	P =   -31.996 deg,	R =    -8.428 deg
   GP2:
	UF : 1, UT : 1,
	J1=   180.000 deg,	J2=  -150.000 deg
};
P[695]{
   GP1:
	UF : 1, UT : 1,		CONFIG : 'N U T, 0, 0, 0',
	X =   606.617  mm,	Y =  -573.857  mm,	Z =   914.233  mm,
	W =    33.386 deg,	P =   -31.996 deg,	R =    -8.428 deg
   GP2:
	UF : 1, UT : 1,
	J1=   180.000 deg,	J2=  -150.000 deg
};
P[696]{
   GP1:
	UF : 1, UT : 1,		CONFIG : 'N U T, 0, 0, 0',
	X =   426.165  mm,	Y =  -510.830  mm,	Z =  1734.717  mm,
	W =    10.103 deg,	P =   -28.621 deg,	R =   -21.273 deg
   GP2:
	UF : 1, UT : 1,
	J1=   180.000 deg,	J2=  -150.000 deg
};
P[697]{
   GP1:
	UF : 1, UT : 1,		CONFIG : 'N U T, 0, 0, 0',
	X =   973.093  mm,	Y =  -950.831  mm,	Z =  1456.444  mm,
	W =     -.010 deg,	P =    45.866 deg,	R =    90.000 deg
   GP2:
	UF : 0, UT : 1,
	J1=   180.000 deg,	J2=   -90.000 deg
};
P[698]{
   GP1:
	UF : 1, UT : 1,		CONFIG : 'N U T, 0, 0, 0',
	X =  1878.092  mm,	Y = -1312.832  mm,	Z =  1256.443  mm,
	W =   -41.810 deg,	P =   -20.894 deg,	R =   -21.724 deg
   GP2:
	UF : 0, UT : 1,
	J1=   180.000 deg,	J2=   -90.000 deg
};
P[699]{
   GP1:
	UF : 1, UT : 1,		CONFIG : 'N U T, 0, 0, 0',
	X =  1944.092  mm,	Y = -1413.832  mm,	Z =  1049.443  mm,
	W =   -42.701 deg,	P =    18.644 deg,	R =    19.122 deg
   GP2:
	UF : 0, UT : 1,
	J1=   180.000 deg,	J2=   -90.000 deg
};
P[700]{
   GP1:
	UF : 1, UT : 1,		CONFIG : 'N U T, 0, 0, 0',
	X =  1905.343  mm,	Y = -1477.017  mm,	Z =  1025.975  mm,
	W =   -39.881 deg,	P =    23.853 deg,	R =    23.904 deg
   GP2:
	UF : 1, UT : 1,
	J1=   180.000 deg,	J2=   -90.000 deg
};
P[701]{
   GP1:
	UF : 1, UT : 1,		CONFIG : 'N U T, 0, 0, 0',
	X =  1932.126  mm,	Y = -1480.053  mm,	Z =  1024.380  mm,
	W =   -43.541 deg,	P =    14.557 deg,	R =    14.831 deg
   GP2:
	UF : 1, UT : 1,
	J1=   180.000 deg,	J2=   -90.000 deg
};
P[702]{
   GP1:
	UF : 1, UT : 1,		CONFIG : 'N U T, 0, 0, 0',
	X =  1967.611  mm,	Y = -1478.561  mm,	Z =  1026.042  mm,
	W =   -43.535 deg,	P =    14.558 deg,	R =    14.822 deg
   GP2:
	UF : 1, UT : 1,
	J1=   180.000 deg,	J2=   -90.000 deg
};
P[703]{
   GP1:
	UF : 1, UT : 1,		CONFIG : 'N U T, 0, 0, 0',
	X =  2000.593  mm,	Y = -1497.735  mm,	Z =  1025.630  mm,
	W =   -43.543 deg,	P =    14.556 deg,	R =   -14.021 deg
   GP2:
	UF : 1, UT : 1,
	J1=   180.000 deg,	J2=   -90.000 deg
};
P[704]{
   GP1:
	UF : 1, UT : 1,		CONFIG : 'N U T, 0, 0, 0',
	X =  2008.768  mm,	Y = -1507.923  mm,	Z =  1025.740  mm,
	W =   -44.808 deg,	P =     8.520 deg,	R =   -27.703 deg
   GP2:
	UF : 1, UT : 1,
	J1=   180.000 deg,	J2=   -90.000 deg
};
P[705]{
   GP1:
	UF : 1, UT : 1,		CONFIG : 'N U T, 0, 0, 0',
	X =  2053.583  mm,	Y = -1389.775  mm,	Z =  1062.551  mm,
	W =   -44.862 deg,	P =     3.961 deg,	R =   -20.537 deg
   GP2:
	UF : 0, UT : 1,
	J1=   180.000 deg,	J2=   -90.000 deg
};
P[706]{
   GP1:
	UF : 1, UT : 1,		CONFIG : 'N U T, 0, 0, 0',
	X =  1878.092  mm,	Y = -1312.832  mm,	Z =  1256.443  mm,
	W =   -41.810 deg,	P =   -20.894 deg,	R =   -21.724 deg
   GP2:
	UF : 0, UT : 1,
	J1=   180.000 deg,	J2=   -90.000 deg
};
P[707]{
   GP1:
